	{attribute 'TcIecLibraryType'}
	{attribute 'external_name' := 'F_VN_PadImageBorderExp_GUID_A5E5D530_2DE0_2D11_697F_7D2919245E82'}
	(* Add padding around the original image borders. (expert function) *)
	FUNCTION F_VN_PadImageBorderExp : HRESULT
	VAR_INPUT
		ipSrcImage	:	ITcVnImage;	(* Source image *)
		ipPaddedImage	:	REFERENCE TO ITcVnImage;	(* Padded destination image (Same type as ipSrcImage, an appropriate destination image will be created if required.) *)
		nTopBorder	:	UDINT;	(* Padding height in pixels above top border *)
		nBottomBorder	:	UDINT;	(* Padding height in pixels below bottom border *)
		nLeftBorder	:	UDINT;	(* Padding width in pixels before left border *)
		nRightBorder	:	UDINT;	(* Padding width in pixels after right border *)
		ePaddingType	:	ETcVnBorderInterpolationMethod;	(* Specifies how the pixel values of the padding area are determined *)
	END_VAR
	VAR_IN_OUT
		aPaddingValue	:	TcVnVector4_LREAL;	(* Specifies the padding value if CONSTANT is used *)
	END_VAR
	VAR_INPUT
		hrPrev	:	HRESULT;	(* HRESULT indicating the result of previous operations (If SUCCEEDED(hrPrev) equals false, no operation is executed.) *)
	END_VAR

END_FUNCTION

// Functions/Basic Image Operations/F_VN_ReinterpretUnsupportedImage

	{attribute 'TcIecLibraryType'}
	{attribute 'external_name' := 'F_VN_ReinterpretUnsupportedImage_GUID_9CD6B2BD_CBC3_29A4_6E5B_0352FEEB17E8'}
	(* Reinterpret an unsupported image using additional information. If successful, the image will be of a supported type. *)
	FUNCTION F_VN_ReinterpretUnsupportedImage : HRESULT
	VAR_INPUT
		ipImage	:	ITcVnImage;	(* Image to be reinterpreted *)
		ePixelType	:	ETcVnElementType;	(* Pixel element type to be used for reinterpreting the image data *)
		hrPrev	:	HRESULT;	(* HRESULT indicating the result of previous operations (If SUCCEEDED(hrPrev) equals false, no operation is executed.) *)
	END_VAR

END_FUNCTION

// Functions/Basic Image Operations/F_VN_ResetRoi

	{attribute 'TcIecLibraryType'}
	{attribute 'external_name' := 'F_VN_ResetRoi_GUID_2C50FDC2_0370_20BD_7F54_98DAB1E9EC31'}
	(* Reset the region of interest (ROI) of an image. (After this operation, the ROI is set to the entire image.) *)
	FUNCTION F_VN_ResetRoi : HRESULT
	VAR_INPUT
		ipImage	:	ITcVnImage;	(* Image *)
		hrPrev	:	HRESULT;	(* HRESULT indicating the result of previous operations (If SUCCEEDED(hrPrev) equals false, no operation is executed.) *)
	END_VAR

END_FUNCTION

// Functions/Basic Image Operations/F_VN_SetImageChannel

	{attribute 'TcIecLibraryType'}
	{attribute 'external_name' := 'F_VN_SetImageChannel_GUID_0A11D43B_5EFB_299D_5725_A1931D902C34'}
	(* Sets the specified destination image channel to the values of the specified source image channel. *)
	FUNCTION F_VN_SetImageChannel : HRESULT
	VAR_INPUT
		ipSrcImage	:	ITcVnImage;	(* Source image *)
		ipDestImage	:	REFERENCE TO ITcVnImage;	(* Destination image (An appropriate image will be created if required.) *)
		nSrcChannelIndex	:	UINT;	(* Index of the source image channel *)
		nDestChannelIndex	:	UINT;	(* Index of the destination image channel, which will be replaced by the specified source image channel *)
		hrPrev	:	HRESULT;	(* HRESULT indicating the result of previous operations (If SUCCEEDED(hrPrev) equals false, no operation is executed.) *)
	END_VAR

END_FUNCTION

// Functions/Basic Image Operations/F_VN_SetPixel

	{attribute 'TcIecLibraryType'}
	{attribute 'external_name' := 'F_VN_SetPixel_GUID_8B44FC22_04B7_2DC7_7023_0AD245DB3507'}
	(* Sets a specific pixel. *)
	FUNCTION F_VN_SetPixel : HRESULT
	VAR_INPUT
		ipSrcImage	:	ITcVnImage;	(* Source image *)
	END_VAR
	VAR_IN_OUT
		aValue	:	TcVnVector4_LREAL;	(* The pixel value to set (additional channels are ignored.) *)
	END_VAR
	VAR_INPUT
		nX	:	UDINT;	(* x coordinate of the pixel *)
		nY	:	UDINT;	(* y coordinate of the pixel *)
		hrPrev	:	HRESULT;	(* HRESULT indicating the result of previous operations (If SUCCEEDED(hrPrev) equals false, no operation is executed.) *)
	END_VAR

END_FUNCTION

// Functions/Basic Image Operations/F_VN_SetPixels

	{attribute 'TcIecLibraryType'}
	{attribute 'external_name' := 'F_VN_SetPixels_GUID_FAE3DEC6_6066_2303_76C8_108C64D81E38'}
	(* Sets all pixels of an image to a given value. *)
	FUNCTION F_VN_SetPixels : HRESULT
	VAR_INPUT
		ipDestImage	:	ITcVnImage;	(* Destination image *)
	END_VAR
	VAR_IN_OUT
		aValue	:	TcVnVector4_LREAL;	(* Pixel value *)
	END_VAR
	VAR_INPUT
		hrPrev	:	HRESULT;	(* HRESULT indicating the result of previous operations (If SUCCEEDED(hrPrev) equals false, no operation is executed.) *)
	END_VAR

END_FUNCTION

// Functions/Basic Image Operations/F_VN_SetPixelsExp

	{attribute 'TcIecLibraryType'}
	{attribute 'external_name' := 'F_VN_SetPixelsExp_GUID_45CBC089_464B_2FAF_6251_E594A25ABBA2'}
	(* Sets all pixels of an image to a given value. (expert function) *)
	FUNCTION F_VN_SetPixelsExp : HRESULT
	VAR_INPUT
		ipDestImage	:	ITcVnImage;	(* Destination image *)
	END_VAR
	VAR_IN_OUT
		aValue	:	TcVnVector4_LREAL;	(* Pixel value *)
	END_VAR
	VAR_INPUT
		ipMask	:	ITcVnImage;	(* Mask image *)
		hrPrev	:	HRESULT;	(* HRESULT indicating the result of previous operations (If SUCCEEDED(hrPrev) equals false, no operation is executed.) *)
	END_VAR

END_FUNCTION

// Functions/Basic Image Operations/F_VN_SetRoi

	{attribute 'TcIecLibraryType'}
	{attribute 'external_name' := 'F_VN_SetRoi_GUID_6B5F6ACC_D699_29DC_6ACC_234995C24602'}
	(* Sets a region of interest (ROI) within an image. *)
	FUNCTION F_VN_SetRoi : HRESULT
	VAR_INPUT
		nX	:	UDINT;	(* Left boundary (inclusive 0-based index) *)
		nY	:	UDINT;	(* Upper boundary (inclusive 0-based index) *)
		nWidth	:	UDINT;	(* ROI width *)
		nHeight	:	UDINT;	(* ROI height *)
		ipDestImage	:	ITcVnImage;	(* Destination image *)
		hrPrev	:	HRESULT;	(* HRESULT indicating the result of previous operations (If SUCCEEDED(hrPrev) equals false, no operation is executed.) *)
	END_VAR

END_FUNCTION

// Functions/Basic Image Operations/F_VN_SetRoi_TcVnRectangle_DINT

	{attribute 'TcIecLibraryType'}
	{attribute 'external_name' := 'F_VN_SetRoi_TcVnRectangle_DINT_GUID_351427E6_8825_2F16_7392_DBA0A93C3EA1'}
	(* Sets a region of interest (ROI) within an image. *)
	FUNCTION F_VN_SetRoi_TcVnRectangle_DINT : HRESULT
	VAR_IN_OUT
		stRoi	:	TcVnRectangle_DINT;	(* Region of interest *)
	END_VAR
	VAR_INPUT
		ipDestImage	:	ITcVnImage;	(* Destination image *)
		hrPrev	:	HRESULT;	(* HRESULT indicating the result of previous operations (If SUCCEEDED(hrPrev) equals false, no operation is executed.) *)
	END_VAR

END_FUNCTION

// Functions/Basic Image Operations/F_VN_SetRoi_TcVnRectangle_UDINT

	{attribute 'TcIecLibraryType'}
	{attribute 'external_name' := 'F_VN_SetRoi_TcVnRectangle_UDINT_GUID_602E64BE_2371_25A7_7431_0AE2E6733D33'}
	(* Sets a region of interest (ROI) within an image. *)
	FUNCTION F_VN_SetRoi_TcVnRectangle_UDINT : HRESULT
	VAR_IN_OUT
		stRoi	:	TcVnRectangle_UDINT;	(* Region of interest *)
	END_VAR
	VAR_INPUT
		ipDestImage	:	ITcVnImage;	(* Destination image *)
		hrPrev	:	HRESULT;	(* HRESULT indicating the result of previous operations (If SUCCEEDED(hrPrev) equals false, no operation is executed.) *)
	END_VAR

END_FUNCTION

// Functions/Basic Image Operations/F_VN_SplitImageChannels

	{attribute 'TcIecLibraryType'}
	{attribute 'external_name' := 'F_VN_SplitImageChannels_GUID_A95E5FB7_F301_2632_66A4_8427D601C7CB'}
	(* Split a multi-channel image into multiple single channel images (1 for each source image channel). *)
	FUNCTION F_VN_SplitImageChannels : HRESULT
	VAR_INPUT
		ipSrcImage	:	ITcVnImage;	(* Source image with multiple channels *)
		pDestImages	:	PVOID;	(* Pointer to an array of ITcVnImage (appropriate destination images will be created if required) *)
		nArraySize	:	UINT;	(* Number of pDestImages array elements (array must be >= ipSourceImage channels) *)
		hrPrev	:	HRESULT;	(* HRESULT indicating the result of previous operations (If SUCCEEDED(hrPrev) equals false, no operation is executed.) *)
	END_VAR
	VAR_OUTPUT
		nImageChannels	:	UINT;	(* Actual source image channels *)
	END_VAR

END_FUNCTION

// Functions/Basic Image Operations/F_VN_TransformIntoDisplayableImageExp

	{attribute 'TcIecLibraryType'}
	{attribute 'external_name' := 'F_VN_TransformIntoDisplayableImageExp_GUID_167A9D9F_1F20_2D5B_6C90_35CDA27FBBBC'}
	(* Transform an image into a displayable image. The source image will be released and zeroed while existing destination images will be released and overwritten with the function result. If bAllowDeepCopy equals false, the source image must not be used anywhere else and the transformation is always very fast. Otherwise, if bAllowDeepCopy equals true, a deep copy of the source image might be created if required, which will result in a longer execution time. If you want to use ipSrcImage after this function call, use F_VN_CopyIntoDisplayableImage instead. (expert function) *)
	FUNCTION F_VN_TransformIntoDisplayableImageExp : HRESULT
	VAR_INPUT
		ipSrcImage	:	REFERENCE TO ITcVnImage;	(* Source image *)
		ipDestImage	:	REFERENCE TO ITcVnDisplayableImage;	(* Returns the displayable image *)
		bAllowDeepCopy	:	BOOL;	(* Allow deep image copies, if required *)
		hrPrev	:	HRESULT;	(* HRESULT indicating the result of previous operations (If SUCCEEDED(hrPrev) equals false, no operation is executed.) *)
	END_VAR

END_FUNCTION

// Functions/Container Statistics/F_VN_ContainerAverage

	{attribute 'TcIecLibraryType'}
	{attribute 'external_name' := 'F_VN_ContainerAverage_GUID_AA883F39_9BF3_2D50_47D7_60462300CF21'}
	(* Calculate the average of elements in a container. *)
	FUNCTION F_VN_ContainerAverage : HRESULT
	VAR_INPUT
		ipSrcContainer	:	ITcVnContainer;	(* Source container (Arithmetic, point and vector element types are supported. For points and vectors, the euclidean norm is used.) *)
	END_VAR
	VAR_IN_OUT
		fAverage	:	LREAL;	(* Returns the calculated average value *)
	END_VAR
	VAR_INPUT
		hrPrev	:	HRESULT;	(* HRESULT indicating the result of previous operations (If SUCCEEDED(hrPrev) equals false, no operation is executed.) *)
	END_VAR

END_FUNCTION

// Functions/Container Statistics/F_VN_ContainerAverageElementwise2

	{attribute 'TcIecLibraryType'}
	{attribute 'external_name' := 'F_VN_ContainerAverageElementwise2_GUID_A5968F66_4B6A_2FA7_4E6D_E4702B7B6763'}
	(* Calculate the elementwise average of 2D elements in a container. *)
	FUNCTION F_VN_ContainerAverageElementwise2 : HRESULT
	VAR_INPUT
		ipSrcContainer	:	ITcVnContainer;	(* Source container with 2D points or vectors *)
	END_VAR
	VAR_IN_OUT
		aAverage	:	TcVnVector2_LREAL;	(* Returns the calculated average values *)
	END_VAR
	VAR_INPUT
		hrPrev	:	HRESULT;	(* HRESULT indicating the result of previous operations (If SUCCEEDED(hrPrev) equals false, no operation is executed.) *)
	END_VAR

END_FUNCTION

// Functions/Container Statistics/F_VN_ContainerAverageElementwise3

	{attribute 'TcIecLibraryType'}
	{attribute 'external_name' := 'F_VN_ContainerAverageElementwise3_GUID_40FE5448_4613_25F6_6B44_B58BBFE3E301'}
	(* Calculate the elementwise average of 3D elements in a container. *)
	FUNCTION F_VN_ContainerAverageElementwise3 : HRESULT
	VAR_INPUT
		ipSrcContainer	:	ITcVnContainer;	(* Source container with 3D points or vectors *)
	END_VAR
	VAR_IN_OUT
		aAverage	:	TcVnVector3_LREAL;	(* Returns the calculated average values *)
	END_VAR
	VAR_INPUT
		hrPrev	:	HRESULT;	(* HRESULT indicating the result of previous operations (If SUCCEEDED(hrPrev) equals false, no operation is executed.) *)
	END_VAR

END_FUNCTION

// Functions/Container Statistics/F_VN_ContainerAverageElementwise4

	{attribute 'TcIecLibraryType'}
	{attribute 'external_name' := 'F_VN_ContainerAverageElementwise4_GUID_DEACFB72_F4A2_2C02_42D9_1C2A0DD59263'}
	(* Calculate the elementwise average of 4D elements in a container. *)
	FUNCTION F_VN_ContainerAverageElementwise4 : HRESULT
	VAR_INPUT
		ipSrcContainer	:	ITcVnContainer;	(* Source container with 4D vectors *)
	END_VAR
	VAR_IN_OUT
		aAverage	:	TcVnVector4_LREAL;	(* Returns the calculated average values *)
	END_VAR
	VAR_INPUT
		hrPrev	:	HRESULT;	(* HRESULT indicating the result of previous operations (If SUCCEEDED(hrPrev) equals false, no operation is executed.) *)
	END_VAR

END_FUNCTION

// Functions/Container Statistics/F_VN_ContainerAverageVariance

	{attribute 'TcIecLibraryType'}
	{attribute 'external_name' := 'F_VN_ContainerAverageVariance_GUID_F86D5373_0B69_212E_4923_C1F41E37B181'}
	(* Calculate the average and variance of elements in a container. *)
	FUNCTION F_VN_ContainerAverageVariance : HRESULT
	VAR_INPUT
		ipSrcContainer	:	ITcVnContainer;	(* Source container (Arithmetic, point and vector element types are supported. For points and vectors, the euclidean norm is used.) *)
	END_VAR
	VAR_IN_OUT
		fAverage	:	LREAL;	(* Returns the calculated average value *)
		fVariance	:	LREAL;	(* Returns the calculated variance value *)
	END_VAR
	VAR_INPUT
		hrPrev	:	HRESULT;	(* HRESULT indicating the result of previous operations (If SUCCEEDED(hrPrev) equals false, no operation is executed.) *)
	END_VAR

END_FUNCTION

// Functions/Container Statistics/F_VN_ContainerAverageVarianceElementwise2

	{attribute 'TcIecLibraryType'}
	{attribute 'external_name' := 'F_VN_ContainerAverageVarianceElementwise2_GUID_9DD8D138_D087_2ADB_447F_BCA5C1C4B858'}
	(* Calculate the elementwise average and variance of 2D elements in a container. *)
	FUNCTION F_VN_ContainerAverageVarianceElementwise2 : HRESULT
	VAR_INPUT
		ipSrcContainer	:	ITcVnContainer;	(* Source container with 2D points or vectors *)
	END_VAR
	VAR_IN_OUT
		aAverage	:	TcVnVector2_LREAL;	(* Returns the calculated average values *)
		aVariance	:	TcVnVector2_LREAL;	(* Returns the calculated variance values *)
	END_VAR
	VAR_INPUT
		hrPrev	:	HRESULT;	(* HRESULT indicating the result of previous operations (If SUCCEEDED(hrPrev) equals false, no operation is executed.) *)
	END_VAR

END_FUNCTION

// Functions/Container Statistics/F_VN_ContainerAverageVarianceElementwise3

	{attribute 'TcIecLibraryType'}
	{attribute 'external_name' := 'F_VN_ContainerAverageVarianceElementwise3_GUID_FA835F97_60F3_2236_51E3_712391145764'}
	(* Calculate the elementwise average and variance of 3D elements in a container. *)
	FUNCTION F_VN_ContainerAverageVarianceElementwise3 : HRESULT
	VAR_INPUT
		ipSrcContainer	:	ITcVnContainer;	(* Source container with 3D points or vectors *)
	END_VAR
	VAR_IN_OUT
		aAverage	:	TcVnVector3_LREAL;	(* Returns the calculated average values *)
		aVariance	:	TcVnVector3_LREAL;	(* Returns the calculated variance values *)
	END_VAR
	VAR_INPUT
		hrPrev	:	HRESULT;	(* HRESULT indicating the result of previous operations (If SUCCEEDED(hrPrev) equals false, no operation is executed.) *)
	END_VAR

END_FUNCTION

// Functions/Container Statistics/F_VN_ContainerAverageVarianceElementwise4

	{attribute 'TcIecLibraryType'}
	{attribute 'external_name' := 'F_VN_ContainerAverageVarianceElementwise4_GUID_031E1C0B_D296_2CEF_785B_2052A4B44928'}
	(* Calculate the elementwise average and variance of 4D elements in a container. *)
	FUNCTION F_VN_ContainerAverageVarianceElementwise4 : HRESULT
	VAR_INPUT
		ipSrcContainer	:	ITcVnContainer;	(* Source container with 4D vectors *)
	END_VAR
	VAR_IN_OUT
		aAverage	:	TcVnVector4_LREAL;	(* Returns the calculated average values *)
		aVariance	:	TcVnVector4_LREAL;	(* Returns the calculated variance values *)
	END_VAR
	VAR_INPUT
		hrPrev	:	HRESULT;	(* HRESULT indicating the result of previous operations (If SUCCEEDED(hrPrev) equals false, no operation is executed.) *)
	END_VAR

END_FUNCTION

// Functions/Container Statistics/F_VN_MaxElement

	{attribute 'TcIecLibraryType'}
	{attribute 'external_name' := 'F_VN_MaxElement_GUID_9353BD58_8969_23CD_6837_1D5672DD3636'}
	(* Gets the maximum element of a container. *)
	FUNCTION F_VN_MaxElement : HRESULT
	VAR_INPUT
		ipSrcContainer	:	ITcVnContainer;	(* Source container (Arithmetic, point and vector element types are supported. For points and vectors, the euclidean norm is used.) *)
		ipDestIterator	:	REFERENCE TO ITcVnBidirectionalIterator;	(* Returns an iterator to the requested element *)
	END_VAR
	VAR_IN_OUT
		nIndex	:	ULINT;	(* Returns the position of the requested element within the container *)
	END_VAR
	VAR_INPUT
		hrPrev	:	HRESULT;	(* HRESULT indicating the result of previous operations (If SUCCEEDED(hrPrev) equals false, no operation is executed.) *)
	END_VAR

END_FUNCTION

// Functions/Container Statistics/F_VN_MedianElement

	{attribute 'TcIecLibraryType'}
	{attribute 'external_name' := 'F_VN_MedianElement_GUID_734602DB_9D28_2D88_734A_BDC3C8FE153F'}
	(* Gets the median element of a container. *)
	FUNCTION F_VN_MedianElement : HRESULT
	VAR_INPUT
		ipSrcContainer	:	ITcVnContainer;	(* Source container (Arithmetic, point and vector element types are supported. For points and vectors, the euclidean norm is used.) *)
		ipDestIterator	:	REFERENCE TO ITcVnBidirectionalIterator;	(* Returns an iterator to the requested element *)
	END_VAR
	VAR_IN_OUT
		nIndex	:	ULINT;	(* Returns the position of the requested element within the container *)
	END_VAR
	VAR_INPUT
		hrPrev	:	HRESULT;	(* HRESULT indicating the result of previous operations (If SUCCEEDED(hrPrev) equals false, no operation is executed.) *)
	END_VAR

END_FUNCTION

// Functions/Container Statistics/F_VN_MinElement

	{attribute 'TcIecLibraryType'}
	{attribute 'external_name' := 'F_VN_MinElement_GUID_9563E038_8D44_21FD_4C05_B15238CF2018'}
	(* Gets the minimum element of a container. *)
	FUNCTION F_VN_MinElement : HRESULT
	VAR_INPUT
		ipSrcContainer	:	ITcVnContainer;	(* Source container (Arithmetic, point and vector element types are supported. For points and vectors, the euclidean norm is used.) *)
		ipDestIterator	:	REFERENCE TO ITcVnBidirectionalIterator;	(* Returns an iterator to the requested element *)
	END_VAR
	VAR_IN_OUT
		nIndex	:	ULINT;	(* Returns the position of the requested element within the container *)
	END_VAR
	VAR_INPUT
		hrPrev	:	HRESULT;	(* HRESULT indicating the result of previous operations (If SUCCEEDED(hrPrev) equals false, no operation is executed.) *)
	END_VAR

END_FUNCTION

// Functions/Fourier Analysis/F_VN_CreateBandpassButterworthFilter

	{attribute 'TcIecLibraryType'}
	{attribute 'external_name' := 'F_VN_CreateBandpassButterworthFilter_GUID_A4719FC8_3078_205C_4E26_9139901FC7B0'}
	(* Creates a bandpass Butterworth filter, which can be applied to a frequency domain image by element-wise multiplication. *)
	FUNCTION F_VN_CreateBandpassButterworthFilter : HRESULT
	VAR_INPUT
		ipFilter	:	REFERENCE TO ITcVnImage;	(* Returns the created filter (1 channel of type REAL or LREAL, depending on bDoublePrecision. Non-zero interface pointers are reused.). *)
		nWidth	:	UDINT;	(* Filter width (even, >= 2, must match the width of the image it is applied to) *)
		nHeight	:	UDINT;	(* Filter height (even, >= 2, must match the height of the image it is applied to) *)
		bDoublePrecision	:	BOOL;	(* If true, the filter is generated with double precision (LREAL) instead of single precision (REAL). *)
		bOriginAtCenter	:	BOOL;	(* If true, the filter origin is shifted to the image center. *)
		fCutoffDistance	:	LREAL;	(* The cutoff distance of the Butterworth filter (> 0). *)
		fBandWidth	:	LREAL;	(* The band width of the Butterworth filter (> 0). *)
		nOrder	:	UDINT;	(* The order of the Butterworth filter (> 0). *)
		fScale	:	LREAL;	(* The scale factor of the Butterworth filter denominator term (> 0, e.g. 0.414 or 1.0). *)
		hrPrev	:	HRESULT;	(* HRESULT indicating the result of previous operations (If SUCCEEDED(hrPrev) equals false, no operation is executed.) *)
	END_VAR

END_FUNCTION

// Functions/Fourier Analysis/F_VN_CreateBandpassGaussianFilter

	{attribute 'TcIecLibraryType'}
	{attribute 'external_name' := 'F_VN_CreateBandpassGaussianFilter_GUID_AB3E0B05_028B_2322_7CF4_87504E4D004F'}
	(* Creates a bandpass Gaussian filter, which can be applied to a frequency domain image by element-wise multiplication. *)
	FUNCTION F_VN_CreateBandpassGaussianFilter : HRESULT
	VAR_INPUT
		ipFilter	:	REFERENCE TO ITcVnImage;	(* Returns the created filter (1 channel of type REAL or LREAL, depending on bDoublePrecision. Non-zero interface pointers are reused.). *)
		nWidth	:	UDINT;	(* Filter width (even, >= 2, must match the width of the image it is applied to) *)
		nHeight	:	UDINT;	(* Filter height (even, >= 2, must match the height of the image it is applied to) *)
		bDoublePrecision	:	BOOL;	(* If true, the filter is generated with double precision (LREAL) instead of single precision (REAL). *)
		bOriginAtCenter	:	BOOL;	(* If true, the filter origin is shifted to the image center. *)
		fCutoffDistance	:	LREAL;	(* The cutoff distance of the Gaussian filter (> 0). *)
		fBandWidth	:	LREAL;	(* The band width of the Gaussian filter (> 0). *)
		hrPrev	:	HRESULT;	(* HRESULT indicating the result of previous operations (If SUCCEEDED(hrPrev) equals false, no operation is executed.) *)
	END_VAR

END_FUNCTION

// Functions/Fourier Analysis/F_VN_CreateBandrejectButterworthFilter

	{attribute 'TcIecLibraryType'}
	{attribute 'external_name' := 'F_VN_CreateBandrejectButterworthFilter_GUID_43FD0880_9A03_21BB_62EE_0C372A51F6F1'}
	(* Creates a bandreject Butterworth filter, which can be applied to a frequency domain image by element-wise multiplication. *)
	FUNCTION F_VN_CreateBandrejectButterworthFilter : HRESULT
	VAR_INPUT
		ipFilter	:	REFERENCE TO ITcVnImage;	(* Returns the created filter (1 channel of type REAL or LREAL, depending on bDoublePrecision. Non-zero interface pointers are reused.). *)
		nWidth	:	UDINT;	(* Filter width (even, >= 2, must match the width of the image it is applied to) *)
		nHeight	:	UDINT;	(* Filter height (even, >= 2, must match the height of the image it is applied to) *)
		bDoublePrecision	:	BOOL;	(* If true, the filter is generated with double precision (LREAL) instead of single precision (REAL). *)
		bOriginAtCenter	:	BOOL;	(* If true, the filter origin is shifted to the image center. *)
		fCutoffDistance	:	LREAL;	(* The cutoff distance of the Butterworth filter (> 0). *)
		fBandWidth	:	LREAL;	(* The band width of the Butterworth filter (> 0). *)
		nOrder	:	UDINT;	(* The order of the Butterworth filter (> 0). *)
		fScale	:	LREAL;	(* The scale factor of the Butterworth filter denominator term (> 0, e.g. 0.414 or 1.0). *)
		hrPrev	:	HRESULT;	(* HRESULT indicating the result of previous operations (If SUCCEEDED(hrPrev) equals false, no operation is executed.) *)
	END_VAR

END_FUNCTION

// Functions/Fourier Analysis/F_VN_CreateBandrejectGaussianFilter

	{attribute 'TcIecLibraryType'}
	{attribute 'external_name' := 'F_VN_CreateBandrejectGaussianFilter_GUID_2D030AC7_64BE_238B_728C_49B2827F9032'}
	(* Creates a bandreject Gaussian filter, which can be applied to a frequency domain image by element-wise multiplication. *)
	FUNCTION F_VN_CreateBandrejectGaussianFilter : HRESULT
	VAR_INPUT
		ipFilter	:	REFERENCE TO ITcVnImage;	(* Returns the created filter (1 channel of type REAL or LREAL, depending on bDoublePrecision. Non-zero interface pointers are reused.). *)
		nWidth	:	UDINT;	(* Filter width (even, >= 2, must match the width of the image it is applied to) *)
		nHeight	:	UDINT;	(* Filter height (even, >= 2, must match the height of the image it is applied to) *)
		bDoublePrecision	:	BOOL;	(* If true, the filter is generated with double precision (LREAL) instead of single precision (REAL). *)
		bOriginAtCenter	:	BOOL;	(* If true, the filter origin is shifted to the image center. *)
		fCutoffDistance	:	LREAL;	(* The cutoff distance of the Gaussian filter (> 0). *)
		fBandWidth	:	LREAL;	(* The band width of the Gaussian filter (> 0). *)
		hrPrev	:	HRESULT;	(* HRESULT indicating the result of previous operations (If SUCCEEDED(hrPrev) equals false, no operation is executed.) *)
	END_VAR

END_FUNCTION

// Functions/Fourier Analysis/F_VN_CreateHighpassButterworthFilter

	{attribute 'TcIecLibraryType'}
	{attribute 'external_name' := 'F_VN_CreateHighpassButterworthFilter_GUID_26315EFD_6407_2DDF_6510_E1ECDEDCA359'}
	(* Creates a highpass Butterworth filter, which can be applied to a frequency domain image by element-wise multiplication. *)
	FUNCTION F_VN_CreateHighpassButterworthFilter : HRESULT
	VAR_INPUT
		ipFilter	:	REFERENCE TO ITcVnImage;	(* Returns the created filter (1 channel of type REAL or LREAL, depending on bDoublePrecision. Non-zero interface pointers are reused.). *)
		nWidth	:	UDINT;	(* Filter width (even, >= 2, must match the width of the image it is applied to) *)
		nHeight	:	UDINT;	(* Filter height (even, >= 2, must match the height of the image it is applied to) *)
		bDoublePrecision	:	BOOL;	(* If true, the filter is generated with double precision (LREAL) instead of single precision (REAL). *)
		bOriginAtCenter	:	BOOL;	(* If true, the filter origin is shifted to the image center. *)
		fCutoffDistance	:	LREAL;	(* The cutoff distance of the Butterworth filter (> 0). *)
		nOrder	:	UDINT;	(* The order of the Butterworth filter (> 0). *)
		fScale	:	LREAL;	(* The scale factor of the Butterworth filter denominator term (> 0, e.g. 0.414 or 1.0). *)
		hrPrev	:	HRESULT;	(* HRESULT indicating the result of previous operations (If SUCCEEDED(hrPrev) equals false, no operation is executed.) *)
	END_VAR

END_FUNCTION

// Functions/Fourier Analysis/F_VN_CreateHighpassGaussianFilter

	{attribute 'TcIecLibraryType'}
	{attribute 'external_name' := 'F_VN_CreateHighpassGaussianFilter_GUID_91B5C0DC_EE24_21D2_4440_C5D5A4FE32A8'}
	(* Creates a highpass Gaussian filter, which can be applied to a frequency domain image by element-wise multiplication. *)
	FUNCTION F_VN_CreateHighpassGaussianFilter : HRESULT
	VAR_INPUT
		ipFilter	:	REFERENCE TO ITcVnImage;	(* Returns the created filter (1 channel of type REAL or LREAL, depending on bDoublePrecision. Non-zero interface pointers are reused.). *)
		nWidth	:	UDINT;	(* Filter width (even, >= 2, must match the width of the image it is applied to) *)
		nHeight	:	UDINT;	(* Filter height (even, >= 2, must match the height of the image it is applied to) *)
		bDoublePrecision	:	BOOL;	(* If true, the filter is generated with double precision (LREAL) instead of single precision (REAL). *)
		bOriginAtCenter	:	BOOL;	(* If true, the filter origin is shifted to the image center. *)
		fCutoffDistance	:	LREAL;	(* The cutoff distance of the Gaussian filter (> 0). *)
		hrPrev	:	HRESULT;	(* HRESULT indicating the result of previous operations (If SUCCEEDED(hrPrev) equals false, no operation is executed.) *)
	END_VAR

END_FUNCTION

// Functions/Fourier Analysis/F_VN_CreateLowpassButterworthFilter

	{attribute 'TcIecLibraryType'}
	{attribute 'external_name' := 'F_VN_CreateLowpassButterworthFilter_GUID_373093B4_3E27_26A4_696A_3EE89B988877'}
	(* Creates a lowpass Butterworth filter, which can be applied to a frequency domain image by element-wise multiplication. *)
	FUNCTION F_VN_CreateLowpassButterworthFilter : HRESULT
	VAR_INPUT
		ipFilter	:	REFERENCE TO ITcVnImage;	(* Returns the created filter (1 channel of type REAL or LREAL, depending on bDoublePrecision. Non-zero interface pointers are reused.). *)
		nWidth	:	UDINT;	(* Filter width (even, >= 2, must match the width of the image it is applied to) *)
		nHeight	:	UDINT;	(* Filter height (even, >= 2, must match the height of the image it is applied to) *)
		bDoublePrecision	:	BOOL;	(* If true, the filter is generated with double precision (LREAL) instead of single precision (REAL). *)
		bOriginAtCenter	:	BOOL;	(* If true, the filter origin is shifted to the image center. *)
		fCutoffDistance	:	LREAL;	(* The cutoff distance of the Butterworth filter (> 0). *)
		nOrder	:	UDINT;	(* The order of the Butterworth filter (> 0). *)
		fScale	:	LREAL;	(* The scale factor of the Butterworth filter denominator term (> 0, e.g. 0.414 or 1.0). *)
		hrPrev	:	HRESULT;	(* HRESULT indicating the result of previous operations (If SUCCEEDED(hrPrev) equals false, no operation is executed.) *)
	END_VAR

END_FUNCTION

// Functions/Fourier Analysis/F_VN_CreateLowpassGaussianFilter

	{attribute 'TcIecLibraryType'}
	{attribute 'external_name' := 'F_VN_CreateLowpassGaussianFilter_GUID_FC365988_00B2_289F_4A02_DA34E2899A69'}
	(* Creates a lowpass Gaussian filter, which can be applied to a frequency domain image by element-wise multiplication. *)
	FUNCTION F_VN_CreateLowpassGaussianFilter : HRESULT
	VAR_INPUT
		ipFilter	:	REFERENCE TO ITcVnImage;	(* Returns the created filter (1 channel of type REAL or LREAL, depending on bDoublePrecision. Non-zero interface pointers are reused.). *)
		nWidth	:	UDINT;	(* Filter width (even, >= 2, must match the width of the image it is applied to) *)
		nHeight	:	UDINT;	(* Filter height (even, >= 2, must match the height of the image it is applied to) *)
		bDoublePrecision	:	BOOL;	(* If true, the filter is generated with double precision (LREAL) instead of single precision (REAL). *)
		bOriginAtCenter	:	BOOL;	(* If true, the filter origin is shifted to the image center. *)
		fCutoffDistance	:	LREAL;	(* The cutoff distance of the Gaussian filter (> 0). *)
		hrPrev	:	HRESULT;	(* HRESULT indicating the result of previous operations (If SUCCEEDED(hrPrev) equals false, no operation is executed.) *)
	END_VAR

END_FUNCTION

// Functions/Fourier Analysis/F_VN_Dft

	{attribute 'TcIecLibraryType'}
	{attribute 'external_name' := 'F_VN_Dft_GUID_9CD2E68A_8224_2AA6_4C68_735CDE258796'}
	(* Computes the DFT for a given image. *)
	FUNCTION F_VN_Dft : HRESULT
	VAR_INPUT
		ipSpatialImage	:	ITcVnImage;	(* Source image (elements of type REAL or LREAL, 1 (Re) or 2 (Re + Im) channels) *)
		ipFrequencyImage	:	REFERENCE TO ITcVnImage;	(* Destination image (same type as ipSpatialImage, but number of channels and size can vary depending on bPackedCCS and bAutoPadding. *)
		bPackedCCS	:	BOOL;	(* If true and ipSpatialImage has only 1 channel, the result image will have 1 channel with packed complex-conjugate-symmetrical format results. Otherwise, the result image will have 2 separate channels (Re + Im), containing the full spectrum. *)
		bAutoPadding	:	BOOL;	(* If true, the input image is automatically padded (with 0s) to optimal size if required, to speed up dft (Creates a temporary copy so that ipSpatialImage content stays unchanged, which also requires some additional computation power. Therefore, it is recommended to compare execution times with and without padding.) *)
		hrPrev	:	HRESULT;	(* HRESULT indicating the result of previous operations (If SUCCEEDED(hrPrev) equals false, no operation is executed.) *)
	END_VAR

END_FUNCTION

// Functions/Fourier Analysis/F_VN_InverseDft

	{attribute 'TcIecLibraryType'}
	{attribute 'external_name' := 'F_VN_InverseDft_GUID_5190C4B2_3FA3_2B1D_6D96_EBC870B13024'}
	(* Compute the inverse DFT for a given frequency image. *)
	FUNCTION F_VN_InverseDft : HRESULT
	VAR_INPUT
		ipFrequencyImage	:	ITcVnImage;	(* Source frequency image (elements of type REAL or LREAL, 1 (packed CCS) or 2 (Re + Im) channels) *)
		ipSpatialImage	:	REFERENCE TO ITcVnImage;	(* Destination image (Same type as ipFrequencyImage, but number of channels can vary depending on bRealOutput. An appropriate image will be created if required.) *)
		bRealOutput	:	BOOL;	(* Only relevant if ipFrequencyImage has 2 channels. If true, the result image will have only 1 channel. Otherwise, the result image will have 2 separate channels (Re + Im). If ipFrequencyImage has only 1 channel, packed CCS format is assumed and the result image will always have only 1 channel. *)
		hrPrev	:	HRESULT;	(* HRESULT indicating the result of previous operations (If SUCCEEDED(hrPrev) equals false, no operation is executed.) *)
	END_VAR

END_FUNCTION

// Functions/Fourier Analysis/F_VN_OptimalDftSize

	{attribute 'TcIecLibraryType'}
	{attribute 'external_name' := 'F_VN_OptimalDftSize_GUID_7F72AB5E_E31E_25EC_575C_20FDDD4E5230'}
	(* Computes the optimal image size for applying a dft (can lead to better performance). *)
	FUNCTION F_VN_OptimalDftSize : HRESULT
	VAR_INPUT
		ipImage	:	ITcVnImage;	(* Source image for which to compute the optimal width and height *)
	END_VAR
	VAR_IN_OUT
		nOptWidth	:	UDINT;	(* Returns the optimal width of the image *)
		nOptHeight	:	UDINT;	(* Returns the optimal height of the image *)
	END_VAR
	VAR_INPUT
		hrPrev	:	HRESULT;	(* HRESULT indicating the result of previous operations (If SUCCEEDED(hrPrev) equals false, no operation is executed.) *)
	END_VAR

END_FUNCTION

// Functions/Machine Learning/F_VN_CreateBoostClassifier

	{attribute 'TcIecLibraryType'}
	{attribute 'external_name' := 'F_VN_CreateBoostClassifier_GUID_DE956DB3_C6B5_20EF_6F40_CA0A52E7B053'}
	(* Create a Boost classifier using the default parameters. The initial reference count is set to one if a new model is created and kept, otherwise. The Boost classifier is only applicable to binary classification problems. It learns to distinguish between samples labelled with two user-defined class labels by incrementally adding weak classifiers to improve the classification results. Models of this type neither support on-line training (sample by sample) nor retraining. *)
	FUNCTION F_VN_CreateBoostClassifier : HRESULT
	VAR_INPUT
		ipMlModel	:	REFERENCE TO ITcVnMlModel;	(* Returns the created model (Non-zero interface pointers are reused.) *)
		hrPrev	:	HRESULT;	(* HRESULT indicating the result of previous operations (If SUCCEEDED(hrPrev) equals false, no operation is executed.) *)
	END_VAR

END_FUNCTION

// Functions/Machine Learning/F_VN_CreateBoostClassifierExp

	{attribute 'TcIecLibraryType'}
	{attribute 'external_name' := 'F_VN_CreateBoostClassifierExp_GUID_DBB0D30D_27D6_284A_7AD2_009715990AF3'}
	(* Create a Boost classifier. The initial reference count is set to one if a new model is created and kept, otherwise. The Boost classifier is only applicable to binary classification problems. It learns to distinguish between samples labelled with two user-defined class labels by incrementally adding weak classifiers to improve the classification results. Models of this type neither support on-line training (sample by sample) nor retraining. (expert function) *)
	FUNCTION F_VN_CreateBoostClassifierExp : HRESULT
	VAR_INPUT
		ipMlModel	:	REFERENCE TO ITcVnMlModel;	(* Returns the created model (Non-zero interface pointers are reused.) *)
		eType	:	ETcVnBoostClassifierType;	(* Learning algorithm type (default: TCVN_BCT_REAL) *)
		nMaxDepth	:	UDINT;	(* Maximum tree depth (default: 1) *)
		nMinSamples	:	UDINT;	(* Minimum number of samples within a node required for splitting (default: 10) *)
		nWeakClassifiers	:	UDINT;	(* Number of weak classifiers (default: 100) *)
		fWeightTrimRate	:	LREAL;	(* Weight threshold used during training (off: 0; default: 0.95). *)
		hrPrev	:	HRESULT;	(* HRESULT indicating the result of previous operations (If SUCCEEDED(hrPrev) equals false, no operation is executed.) *)
	END_VAR

END_FUNCTION

// Functions/Machine Learning/F_VN_CreateBoostClassifierExp2

	{attribute 'TcIecLibraryType'}
	{attribute 'external_name' := 'F_VN_CreateBoostClassifierExp2_GUID_6FAFAEAC_CC9F_2757_6896_43BC81C44B2C'}
	(* Create a Boost classifier. The initial reference count is set to one if a new model is created and kept, otherwise. The Boost classifier is only applicable to binary classification problems. It learns to distinguish between samples labelled with two user-defined class labels by incrementally adding weak classifiers to improve the classification results. Models of this type neither support on-line training (sample by sample) nor retraining. (expert function) *)
	FUNCTION F_VN_CreateBoostClassifierExp2 : HRESULT
	VAR_INPUT
		ipMlModel	:	REFERENCE TO ITcVnMlModel;	(* Returns the created model (Non-zero interface pointers are reused.) *)
		eType	:	ETcVnBoostClassifierType;	(* Learning algorithm type (default: TCVN_BCT_REAL) *)
		nMaxDepth	:	UDINT;	(* Maximum tree depth (default: 1) *)
		nMinSamples	:	UDINT;	(* Minimum number of samples within a node required for splitting (default: 10) *)
		nWeakClassifiers	:	UDINT;	(* Number of weak classifiers (default: 100) *)
		fWeightTrimRate	:	LREAL;	(* Weight threshold used during training (off: 0; default: 0.95). *)
		ipClassPriors	:	ITcVnContainer;	(* Class priors (ContainerType_Vector_REAL or ContainerType_Vector_LREAL; only for classifiers; optional, set to 0 if not required or not allowed; default: 0) *)
		hrPrev	:	HRESULT;	(* HRESULT indicating the result of previous operations (If SUCCEEDED(hrPrev) equals false, no operation is executed.) *)
	END_VAR

END_FUNCTION

// Functions/Machine Learning/F_VN_CreateKmppModel

	{attribute 'TcIecLibraryType'}
	{attribute 'external_name' := 'F_VN_CreateKmppModel_GUID_FC31DC4A_EF37_2F62_55C6_7F765B594AB6'}
	(* Create a k-means++ model of the specified type. The initial reference count is set to one if a new model is created and kept, otherwise. Models of this type neither support on-line training (sample by sample) nor retraining. *)
	FUNCTION F_VN_CreateKmppModel : HRESULT
	VAR_INPUT
		ipMlModel	:	REFERENCE TO ITcVnMlModel;	(* Returns the created model (Non-zero interface pointers are reused.) *)
		eKmppType	:	ETcVnPrototypeClusterer;	(* k-means++ model type *)
		nK	:	UDINT;	(* Parameter k (number of clusters) *)
		hrPrev	:	HRESULT;	(* HRESULT indicating the result of previous operations (If SUCCEEDED(hrPrev) equals false, no operation is executed.) *)
	END_VAR

END_FUNCTION

// Functions/Machine Learning/F_VN_CreateKmppModelExp

	{attribute 'TcIecLibraryType'}
	{attribute 'external_name' := 'F_VN_CreateKmppModelExp_GUID_91671E6C_0B95_2041_7EBD_EB43C5B888BE'}
	(* Create a k-means++ model of the specified type. The initial reference count is set to one if a new model is created and kept, otherwise. Models of this type neither support on-line training (sample by sample) nor retraining. (expert function) *)
	FUNCTION F_VN_CreateKmppModelExp : HRESULT
	VAR_INPUT
		ipMlModel	:	REFERENCE TO ITcVnMlModel;	(* Returns the created model (Non-zero interface pointers are reused.) *)
		eKmppType	:	ETcVnPrototypeClusterer;	(* k-means++ model type *)
		nK	:	UDINT;	(* Parameter k (number of clusters) *)
		bDoublePrecision	:	BOOL;	(* If true, the model is generated with double precision (LREAL) instead of single precision (REAL). (default: FALSE) *)
		nMaxIterations	:	UDINT;	(* Maximum number of iterations (triggers the usage of the default value of 10 if it equals 0) *)
		fEpsilon	:	LREAL;	(* Maximum allowed difference of the error between two successive iterations (triggers the usage of the default value of 0.001 if it equals 0) *)
		hrPrev	:	HRESULT;	(* HRESULT indicating the result of previous operations (If SUCCEEDED(hrPrev) equals false, no operation is executed.) *)
	END_VAR

END_FUNCTION

// Functions/Machine Learning/F_VN_CreateKnnModel

	{attribute 'TcIecLibraryType'}
	{attribute 'external_name' := 'F_VN_CreateKnnModel_GUID_3FC5A2A1_2868_235E_7F18_46CEDDCDBFFE'}
	(* Create a k-nearest neighbors model of the specified type. The initial reference count is set to one if a new model is created and kept, otherwise. Models of this type support on-line training (sample by sample) and retraining. Predictions can only be scalar. *)
	FUNCTION F_VN_CreateKnnModel : HRESULT
	VAR_INPUT
		ipMlModel	:	REFERENCE TO ITcVnMlModel;	(* Returns the created model (Non-zero interface pointers are reused.) *)
		eKnnType	:	ETcVnKnn;	(* k-nearest neighbors model type *)
		nK	:	UDINT;	(* Parameter k used for prediction (number of considered neighbors) *)
		hrPrev	:	HRESULT;	(* HRESULT indicating the result of previous operations (If SUCCEEDED(hrPrev) equals false, no operation is executed.) *)
	END_VAR

END_FUNCTION

// Functions/Machine Learning/F_VN_CreateLbgModel

	{attribute 'TcIecLibraryType'}
	{attribute 'external_name' := 'F_VN_CreateLbgModel_GUID_A89F132A_3261_218A_640A_D3FE962B6F46'}
	(* Create a LBG model of the specified type. The initial reference count is set to one if a new model is created and kept, otherwise. Models of this type neither support on-line training (sample by sample) nor retraining. *)
	FUNCTION F_VN_CreateLbgModel : HRESULT
	VAR_INPUT
		ipMlModel	:	REFERENCE TO ITcVnMlModel;	(* Returns the created model (Non-zero interface pointers are reused.) *)
		eLbgType	:	ETcVnPrototypeClusterer;	(* LBG model type *)
		nMaxClusters	:	UDINT;	(* Maximum number of clusters *)
		fMaxClusterRadius	:	LREAL;	(* Maximum allowed radius (L2 norm) of a single cluster, i.e. clusters with a higher radius will be split into smaller ones, until a global number of nMaxClusters is reached. *)
		bSingleSplitSteps	:	BOOL;	(* If true, the global optimization is always run after a single cluster has been split. If false, several clusters are split within the same step before applying the global optimization. Applying the global optimization less often is faster, but can lead to less optimal results, especially having 2 nearby clusters that could be represented by 1. *)
		hrPrev	:	HRESULT;	(* HRESULT indicating the result of previous operations (If SUCCEEDED(hrPrev) equals false, no operation is executed.) *)
	END_VAR

END_FUNCTION

// Functions/Machine Learning/F_VN_CreateLbgModelExp

	{attribute 'TcIecLibraryType'}
	{attribute 'external_name' := 'F_VN_CreateLbgModelExp_GUID_7D80325A_5FE2_204A_5847_DCDBD3907200'}
	(* Create a LBG model of the specified type. The initial reference count is set to one if a new model is created and kept, otherwise. Models of this type neither support on-line training (sample by sample) nor retraining. (expert function) *)
	FUNCTION F_VN_CreateLbgModelExp : HRESULT
	VAR_INPUT
		ipMlModel	:	REFERENCE TO ITcVnMlModel;	(* Returns the created model (Non-zero interface pointers are reused.) *)
		eLbgType	:	ETcVnPrototypeClusterer;	(* LBG model type *)
		nMaxClusters	:	UDINT;	(* Maximum number of clusters *)
		fMaxClusterRadius	:	LREAL;	(* Maximum allowed radius (L2 norm) of a single cluster, i.e. clusters with a higher radius will be split into smaller ones, until a global number of nMaxClusters is reached. *)
		bSingleSplitSteps	:	BOOL;	(* If true, the global optimization is always run after a single cluster has been split. If false, several clusters are split within the same step before applying the global optimization. Applying the global optimization less often is faster, but can lead to less optimal results, especially having 2 nearby clusters that could be represented by 1. *)
		bDoublePrecision	:	BOOL;	(* If true, the model is generated with double precision (LREAL) instead of single precision (REAL). (default: FALSE) *)
		nMaxIterations	:	UDINT;	(* Maximum number of iterations (triggers the usage of the default value of 10 if it equals 0) *)
		fEpsilon	:	LREAL;	(* Maximum allowed difference of the error between two successive iterations (triggers the usage of the default value of 0.001 if it equals 0) *)
		hrPrev	:	HRESULT;	(* HRESULT indicating the result of previous operations (If SUCCEEDED(hrPrev) equals false, no operation is executed.) *)
	END_VAR

END_FUNCTION

// Functions/Machine Learning/F_VN_CreateLdaTransform

	{attribute 'TcIecLibraryType'}
	{attribute 'external_name' := 'F_VN_CreateLdaTransform_GUID_BFEE6E72_265C_2874_673C_367B017B49AA'}
	(* Create an LDA-based feature transform from the provided data. The number of samples must be >= the number of features and the number of classes must be >= 2. The initial reference count is set to one if a new model is created and kept, otherwise. *)
	FUNCTION F_VN_CreateLdaTransform : HRESULT
	VAR_INPUT
		ipMlModel	:	REFERENCE TO ITcVnMlModel;	(* Returns the created feature transform (Non-zero interface pointers are reused.) *)
		ipSamples	:	ITcUnknown;	(* Container holding a batch of input samples (ContainerType_Vector_Vector_REAL or ContainerType_Vector_Vector_LREAL) *)
		ipClasses	:	ITcVnContainer;	(* Class labels corresponding to the input samples (ContainerType_Vector_DINT) *)
		hrPrev	:	HRESULT;	(* HRESULT indicating the result of previous operations (If SUCCEEDED(hrPrev) equals false, no operation is executed.) *)
	END_VAR

END_FUNCTION

// Functions/Machine Learning/F_VN_CreateLdaTransformViaComponentNum

	{attribute 'TcIecLibraryType'}
	{attribute 'external_name' := 'F_VN_CreateLdaTransformViaComponentNum_GUID_9BEA4391_283A_253A_73D7_A94E3C32FB17'}
	(* Create an LDA-based feature transform from the provided data where the number of components to be used is predefined. The number of samples must be >= the number of features and the number of classes must be >= 2. The initial reference count is set to one if a new model is created and kept, otherwise. (expert function) *)
	FUNCTION F_VN_CreateLdaTransformViaComponentNum : HRESULT
	VAR_INPUT
		ipMlModel	:	REFERENCE TO ITcVnMlModel;	(* Returns the created feature transform (Non-zero interface pointers are reused.) *)
		ipSamples	:	ITcUnknown;	(* Container holding a batch of input samples (ContainerType_Vector_Vector_REAL or ContainerType_Vector_Vector_LREAL) *)
		ipClasses	:	ITcVnContainer;	(* Class labels corresponding to the input samples (ContainerType_Vector_DINT) *)
		nComponentNum	:	UDINT;	(* Number of components (nComponentNum must be smaller than the number of classes. A value of 0 results in the automatic computation of the maximum number of components.) *)
		hrPrev	:	HRESULT;	(* HRESULT indicating the result of previous operations (If SUCCEEDED(hrPrev) equals false, no operation is executed.) *)
	END_VAR

END_FUNCTION

// Functions/Machine Learning/F_VN_CreateNbcModel

	{attribute 'TcIecLibraryType'}
	{attribute 'external_name' := 'F_VN_CreateNbcModel_GUID_DA02C3CE_3432_20F0_76B8_8F9342393153'}
	(* Create a normal Bayes classifier of the specified type. The initial reference count is set to one if a new model is created and kept, otherwise. In order to train normal Bayes classifiers, a sufficiently high number of samples is required for each class. It depends on the number of features and the distribution of the data. Hence, it needs to be tested for each application. Models of this type do not support on-line training (sample by sample). For the retraining of such classifier models, the set of presented classes must be identical to the previous learning steps. Otherwise, an exception is raised. *)
	FUNCTION F_VN_CreateNbcModel : HRESULT
	VAR_INPUT
		ipMlModel	:	REFERENCE TO ITcVnMlModel;	(* Returns the created model (Non-zero interface pointers are reused.) *)
		eNbcType	:	ETcVnNbc;	(* Normal Bayes classifier type *)
		hrPrev	:	HRESULT;	(* HRESULT indicating the result of previous operations (If SUCCEEDED(hrPrev) equals false, no operation is executed.) *)
	END_VAR

END_FUNCTION

// Functions/Machine Learning/F_VN_CreatePcaTransform

	{attribute 'TcIecLibraryType'}
	{attribute 'external_name' := 'F_VN_CreatePcaTransform_GUID_DA24C08E_FFC7_2FDD_40DC_07CC6EFE8395'}
	(* Create a PCA-based feature transform from the provided data. The maximum number of principal components that can be computed equals the minimum of the number of samples and the number of features. The initial reference count is set to one if a new model is created and kept, otherwise. *)
	FUNCTION F_VN_CreatePcaTransform : HRESULT
	VAR_INPUT
		ipMlModel	:	REFERENCE TO ITcVnMlModel;	(* Returns the created feature transform (Non-zero interface pointers are reused.) *)
		ipSamples	:	ITcUnknown;	(* Container holding a batch of input samples (ContainerType_Vector_Vector_REAL or ContainerType_Vector_Vector_LREAL) *)
		hrPrev	:	HRESULT;	(* HRESULT indicating the result of previous operations (If SUCCEEDED(hrPrev) equals false, no operation is executed.) *)
	END_VAR

END_FUNCTION

// Functions/Machine Learning/F_VN_CreatePcaTransformViaComponentNum

	{attribute 'TcIecLibraryType'}
	{attribute 'external_name' := 'F_VN_CreatePcaTransformViaComponentNum_GUID_28104B27_51EA_20F4_57BD_7EF798538D8F'}
	(* Create a PCA-based feature transform from the provided data where the number of prinicpal components to be used is predefined. The maximum number of principal components that can be computed equals the minimum of the number of samples and the number of features. The initial reference count is set to one if a new model is created and kept, otherwise. (expert function) *)
	FUNCTION F_VN_CreatePcaTransformViaComponentNum : HRESULT
	VAR_INPUT
		ipMlModel	:	REFERENCE TO ITcVnMlModel;	(* Returns the created feature transform (Non-zero interface pointers are reused.) *)
		ipSamples	:	ITcUnknown;	(* Container holding a batch of input samples (ContainerType_Vector_Vector_REAL or ContainerType_Vector_Vector_LREAL) *)
		nComponentNum	:	UDINT;	(* Number of principal components (A value of 0 results in the automatic computation of the maximum number of components.) *)
		hrPrev	:	HRESULT;	(* HRESULT indicating the result of previous operations (If SUCCEEDED(hrPrev) equals false, no operation is executed.) *)
	END_VAR

END_FUNCTION

// Functions/Machine Learning/F_VN_CreatePcaTransformViaVariance

	{attribute 'TcIecLibraryType'}
	{attribute 'external_name' := 'F_VN_CreatePcaTransformViaVariance_GUID_1D00BCB6_0F8E_2453_7A66_86E326231A6F'}
	(* Create a PCA-based feature transform from the provided data based on a given fraction of variance to be retained. The maximum number of principal components that can be computed equals the minimum of the number of samples and the number of features. The initial reference count is set to one if a new model is created and kept, otherwise. (expert function) *)
	FUNCTION F_VN_CreatePcaTransformViaVariance : HRESULT
	VAR_INPUT
		ipMlModel	:	REFERENCE TO ITcVnMlModel;	(* Returns the created feature transform (Non-zero interface pointers are reused.) *)
		ipSamples	:	ITcUnknown;	(* Container holding a batch of input samples (ContainerType_Vector_Vector_REAL or ContainerType_Vector_Vector_LREAL) *)
		fRetainedVariance	:	LREAL;	(* Fraction of variance that is to be retained by the PCA (A value of 1.0 signifies 100%.) *)
		hrPrev	:	HRESULT;	(* HRESULT indicating the result of previous operations (If SUCCEEDED(hrPrev) equals false, no operation is executed.) *)
	END_VAR

END_FUNCTION

// Functions/Machine Learning/F_VN_CreateRTreesModel

	{attribute 'TcIecLibraryType'}
	{attribute 'external_name' := 'F_VN_CreateRTreesModel_GUID_5E8D1899_6C3A_2CDF_5A6E_02E699F01A9E'}
	(* Create a random trees model of the specified type. The initial reference count is set to one if a new model is created and kept, otherwise. Models of this type neither support on-line training (sample by sample) nor retraining. Predictions can only be scalar. *)
	FUNCTION F_VN_CreateRTreesModel : HRESULT
	VAR_INPUT
		ipMlModel	:	REFERENCE TO ITcVnMlModel;	(* Returns the created model (Non-zero interface pointers are reused.) *)
		eRTreesType	:	ETcVnRTrees;	(* Random trees model type *)
		hrPrev	:	HRESULT;	(* HRESULT indicating the result of previous operations (If SUCCEEDED(hrPrev) equals false, no operation is executed.) *)
	END_VAR

END_FUNCTION

// Functions/Machine Learning/F_VN_CreateRTreesModelExp

	{attribute 'TcIecLibraryType'}
	{attribute 'external_name' := 'F_VN_CreateRTreesModelExp_GUID_B4393A32_59CB_20BD_6E6F_3D9FC67F97F8'}
	(* Create a random trees model of the specified type. The initial reference count is set to one if a new model is created and kept, otherwise. Models of this type neither support on-line training (sample by sample) nor retraining. Predictions can only be scalar. (expert function) *)
	FUNCTION F_VN_CreateRTreesModelExp : HRESULT
	VAR_INPUT
		ipMlModel	:	REFERENCE TO ITcVnMlModel;	(* Returns the created model (Non-zero interface pointers are reused.) *)
		eRTreesType	:	ETcVnRTrees;	(* Random trees model type *)
		nMaxDepth	:	UDINT;	(* Maximum tree depth (default: 5) *)
		nMinSamples	:	UDINT;	(* Minimum number of samples within a node required for splitting (default: 10) *)
		nActiveVariables	:	UDINT;	(* Number of variables considered for splitting (0 means sqrt(total number of variables); default: 0) *)
		nMaxIterations	:	UDINT;	(* Maximum number of iterations (disabled if it equals 0 and fEpsilon is different from 0.0; triggers the usage of the default value of 50 if nMaxIterations and fEpsilon equal 0) *)
		fEpsilon	:	LREAL;	(* Maximum allowed difference of the error between two successive iterations (disabled if it equals 0.0 and nMaxIterations is different from 0; triggers the usage of the default value of 0.1 if nMaxIterations and fEpsilon equal 0) *)
		hrPrev	:	HRESULT;	(* HRESULT indicating the result of previous operations (If SUCCEEDED(hrPrev) equals false, no operation is executed.) *)
	END_VAR

END_FUNCTION

// Functions/Machine Learning/F_VN_CreateRTreesModelExp2

	{attribute 'TcIecLibraryType'}
	{attribute 'external_name' := 'F_VN_CreateRTreesModelExp2_GUID_CB2A007E_1A54_217F_7384_3FD84203AD44'}
	(* Create a random trees model of the specified type. The initial reference count is set to one if a new model is created and kept, otherwise. Models of this type neither support on-line training (sample by sample) nor retraining. Predictions can only be scalar. (expert function) *)
	FUNCTION F_VN_CreateRTreesModelExp2 : HRESULT
	VAR_INPUT
		ipMlModel	:	REFERENCE TO ITcVnMlModel;	(* Returns the created model (Non-zero interface pointers are reused.) *)
		eRTreesType	:	ETcVnRTrees;	(* Random trees model type *)
		nMaxDepth	:	UDINT;	(* Maximum tree depth (default: 5) *)
		nMinSamples	:	UDINT;	(* Minimum number of samples within a node required for splitting (default: 10) *)
		nActiveVariables	:	UDINT;	(* Number of variables considered for splitting (0 means sqrt(total number of variables); default: 0) *)
		nMaxIterations	:	UDINT;	(* Maximum number of iterations (disabled if it equals 0 and fEpsilon is different from 0.0; triggers the usage of the default value of 50 if nMaxIterations and fEpsilon equal 0) *)
		fEpsilon	:	LREAL;	(* Maximum allowed difference of the error between two successive iterations (disabled if it equals 0.0 and nMaxIterations is different from 0; triggers the usage of the default value of 0.1 if nMaxIterations and fEpsilon equal 0) *)
		fRegressionAccuracy	:	REAL;	(* Termination criterion for regressors (only for regressors; set to default if not allowed; default: 0.0) *)
		ipClassPriors	:	ITcVnContainer;	(* Class priors (ContainerType_Vector_REAL or ContainerType_Vector_LREAL; only for classifiers; optional, set to 0 if not required or not allowed; default: 0) *)
		hrPrev	:	HRESULT;	(* HRESULT indicating the result of previous operations (If SUCCEEDED(hrPrev) equals false, no operation is executed.) *)
	END_VAR

END_FUNCTION

// Functions/Machine Learning/F_VN_CreateStaModel

	{attribute 'TcIecLibraryType'}
	{attribute 'external_name' := 'F_VN_CreateStaModel_GUID_66F6A4E1_5161_2538_5E15_959ACE2242A0'}
	(* Create a Simplified TopoART neural network of the specified type. The initial reference count is set to one if a new model is created and kept, otherwise. Models of this type support on-line training (sample by sample), retraining, as well as scalar and vectorial predictions. It requires all input except class labels (i.e., samples and training outputs/predictions) to lie in the interval [0.0, 1.0]. The predictions of regressors need to be rescaled from the interval [0.0, 1.0] to their respective value range before usage. Depending on the parameter settings and the number of available training samples, repeated training with the same data may improve the results. Like other neural networks based on the Adaptive Resonance Theory (ART), Simplified TopoART neural networks are not prone to catastrophic inference and patricularly well-suited to incremental learning tasks. *)
	FUNCTION F_VN_CreateStaModel : HRESULT
	VAR_INPUT
		ipMlModel	:	REFERENCE TO ITcVnMlModel;	(* Returns the created model (Non-zero interface pointers are reused.) *)
		eStaType	:	ETcVnSta;	(* Simpified TopoART model type *)
		fRho	:	LREAL;	(* Vigilance parameter (controls the number of neurons that are inserted and the maximum size of the formed categories; valid range: [0.0, 1.0]; suggested range: [0.8, 1.0)) *)
		hrPrev	:	HRESULT;	(* HRESULT indicating the result of previous operations (If SUCCEEDED(hrPrev) equals false, no operation is executed.) *)
	END_VAR

END_FUNCTION

// Functions/Machine Learning/F_VN_CreateStaModelExp

	{attribute 'TcIecLibraryType'}
	{attribute 'external_name' := 'F_VN_CreateStaModelExp_GUID_085A0D33_A299_2BF8_4BAF_C8D386BECA2F'}
	(* Create a Simplified TopoART neural network of the specified type. The initial reference count is set to one if a new model is created and kept, otherwise. Models of this type support on-line training (sample by sample), retraining, as well as scalar and vectorial predictions. It requires all input except class labels (i.e., samples and training outputs/predictions) to lie in the interval [0.0, 1.0]. The predictions of regressors need to be rescaled from the interval [0.0, 1.0] to their respective value range before usage. Depending on the parameter settings and the number of available training samples, repeated training with the same data may improve the results. Like other neural networks based on the Adaptive Resonance Theory (ART), Simplified TopoART neural networks are not prone to catastrophic inference and patricularly well-suited to incremental learning tasks. (expert function) *)
	FUNCTION F_VN_CreateStaModelExp : HRESULT
	VAR_INPUT
		ipMlModel	:	REFERENCE TO ITcVnMlModel;	(* Returns the created model (Non-zero interface pointers are reused.) *)
		eStaType	:	ETcVnSta;	(* Simpified TopoART model type *)
		fRho	:	LREAL;	(* Vigilance parameter (controls the number of neurons that are inserted and the maximum size of the formed categories; valid range: [0.0, 1.0]; suggested range: [0.8, 1.0)) *)
		nNu	:	UDINT;	(* Number of neurons used for classification and prediction (must be larger than or equal to 1; suggested range: [1, 10); default: 3) *)
		bDoublePrecision	:	BOOL;	(* If true, the model is generated with double precision (LREAL) instead of single precision (REAL). (default: FALSE) *)
		hrPrev	:	HRESULT;	(* HRESULT indicating the result of previous operations (If SUCCEEDED(hrPrev) equals false, no operation is executed.) *)
	END_VAR

END_FUNCTION

// Functions/Machine Learning/F_VN_CreateStaModelExp2

	{attribute 'TcIecLibraryType'}
	{attribute 'external_name' := 'F_VN_CreateStaModelExp2_GUID_B4C9EC77_862D_2DD5_5390_92D4C6B86CC8'}
	(* Create a Simplified TopoART neural network of the specified type. The initial reference count is set to one if a new model is created and kept, otherwise. Models of this type support on-line training (sample by sample), retraining, as well as scalar and vectorial predictions. It requires all input except class labels (i.e., samples and training outputs/predictions) to lie in the interval [0.0, 1.0]. The predictions of regressors need to be rescaled from the interval [0.0, 1.0] to their respective value range before usage. Depending on the parameter settings and the number of available training samples, repeated training with the same data may improve the results. Like other neural networks based on the Adaptive Resonance Theory (ART), Simplified TopoART neural networks are not prone to catastrophic inference and patricularly well-suited to incremental learning tasks. (additional expert function providing parameters for fine-tuning and noise reduction) *)
	FUNCTION F_VN_CreateStaModelExp2 : HRESULT
	VAR_INPUT
		ipMlModel	:	REFERENCE TO ITcVnMlModel;	(* Returns the created model (Non-zero interface pointers are reused.) *)
		eStaType	:	ETcVnSta;	(* Simpified TopoART model type *)
		fRho	:	LREAL;	(* Vigilance parameter (controls the number of neurons that are inserted and the maximum size of the formed categories; valid range: [0.0, 1.0]; suggested range: [0.8, 1.0)) *)
		nNu	:	UDINT;	(* Number of neurons used for classification and prediction (must be larger than or equal to 1; suggested range: [1, 10); default: 3) *)
		bDoublePrecision	:	BOOL;	(* If true, the model is generated with double precision (LREAL) instead of single precision (REAL). (default: FALSE) *)
		fBetaSbm	:	LREAL;	(* Learning rate of the second best-matching neuron (learning the second best-matching neuron keeps related categories closer together and might improve the results but may require a higher number of neurons and training runs; a value of 0.0 disables learning of the second best-matching neuron; valid range: [0.0, 1.0]; suggested range: [0.0, 0.5]); default: 0.0 *)
		nPhi	:	UDINT;	(* Number of samples a neuron must have learnt to become permanent (required for noise reduction; works in conjunction with nTau; must be larger than or equal to 1; higher values intensify noise reduction; a value of 1 disables removal of neuron candidates; default: 1) *)
		nTau	:	UDINT;	(* Number of learning steps after which node removal is performed (required for noise reduction; works in conjunction with nPhi; must be large enough to allow neuron candidates representing non-noise samples to become the best-matching neuron at least nPhi times before node removal; default: 100) *)
		hrPrev	:	HRESULT;	(* HRESULT indicating the result of previous operations (If SUCCEEDED(hrPrev) equals false, no operation is executed.) *)
	END_VAR

END_FUNCTION

// Functions/Machine Learning/F_VN_CreateSvmModel

	{attribute 'TcIecLibraryType'}
	{attribute 'external_name' := 'F_VN_CreateSvmModel_GUID_0E9B46AA_E9FD_244C_7078_B9DB23BF7170'}
	(* Create an SVM model of the specified type. The initial reference count is set to one if a new model is created and kept, otherwise. Models of this type neither support on-line training (sample by sample) nor retraining. Predictions can only be scalar. *)
	FUNCTION F_VN_CreateSvmModel : HRESULT
	VAR_INPUT
		ipMlModel	:	REFERENCE TO ITcVnMlModel;	(* Returns the created model (Non-zero interface pointers are reused.) *)
		eSvmType	:	ETcVnSvm;	(* SVM model type *)
		fC	:	LREAL;	(* Parameter C (required for TCVN_SVM_C_CLASSIFIER, TCVN_SVM_EPS_REGRESSOR, and TCVN_SVM_NU_REGRESSOR; ignored otherwise) *)
		fNu	:	LREAL;	(* Parameter nu (required for TCVN_SVM_NU_CLASSIFIER, TCVN_SVM_NOVELTY_DETECTOR, and TCVN_SVM_NU_REGRESSOR; ignored otherwise) *)
		fP	:	LREAL;	(* Parameter p (required for TCVN_SVM_EPS_REGRESSOR; ignored otherwise) *)
		eKernelType	:	ETcVnSvmKernelType;	(* Kernel type *)
		fGamma	:	LREAL;	(* Parameter gamma (used by polynomial, RBF, sigmoid, and chi-squared kernels; ignored otherwise) *)
		fCoef0	:	LREAL;	(* parameter coef0 (used by polynomial and sigmoid kernels; ignored otherwise) *)
		fDegree	:	LREAL;	(* Degree (used by polynomial kernels; ignored otherwise) *)
		hrPrev	:	HRESULT;	(* HRESULT indicating the result of previous operations (If SUCCEEDED(hrPrev) equals false, no operation is executed.) *)
	END_VAR

END_FUNCTION

// Functions/Machine Learning/F_VN_CreateSvmModelExp

	{attribute 'TcIecLibraryType'}
	{attribute 'external_name' := 'F_VN_CreateSvmModelExp_GUID_038EDCA5_BA03_2CC3_41B7_ACD066032535'}
	(* Create an SVM model of the specified type. The initial reference count is set to one if a new model is created and kept, otherwise. Models of this type neither support on-line training (sample by sample) nor retraining. Predictions can only be scalar. (expert function) *)
	FUNCTION F_VN_CreateSvmModelExp : HRESULT
	VAR_INPUT
		ipMlModel	:	REFERENCE TO ITcVnMlModel;	(* Returns the created model (Non-zero interface pointers are reused.) *)
		eSvmType	:	ETcVnSvm;	(* SVM model type *)
		fC	:	LREAL;	(* Parameter C (required for TCVN_SVM_C_CLASSIFIER, TCVN_SVM_EPS_REGRESSOR, and TCVN_SVM_NU_REGRESSOR; ignored otherwise) *)
		fNu	:	LREAL;	(* Parameter nu (required for TCVN_SVM_NU_CLASSIFIER, TCVN_SVM_NOVELTY_DETECTOR, and TCVN_SVM_NU_REGRESSOR; ignored otherwise) *)
		fP	:	LREAL;	(* Parameter p (required for TCVN_SVM_EPS_REGRESSOR; ignored otherwise) *)
		eKernelType	:	ETcVnSvmKernelType;	(* Kernel type *)
		fGamma	:	LREAL;	(* Parameter gamma (used by polynomial, RBF, sigmoid, and chi-squared kernels; ignored otherwise) *)
		fCoef0	:	LREAL;	(* Parameter coef0 (used by polynomial and sigmoid kernels; ignored otherwise) *)
		fDegree	:	LREAL;	(* Degree (used by polynomial kernels; ignored otherwise) *)
		nMaxIterations	:	UDINT;	(* Maximum number of iterations (disabled if it equals 0 and fEpsilon is different from 0.0; triggers the usage of the default value of 100000 if nMaxIterations and fEpsilon equal 0) *)
		fEpsilon	:	LREAL;	(* Maximum allowed difference of the error between two successive iterations (disabled if it equals 0.0 and nMaxIterations is different from 0; triggers the usage of the default value of 0.00001 if nMaxIterations and fEpsilon equal 0) *)
		hrPrev	:	HRESULT;	(* HRESULT indicating the result of previous operations (If SUCCEEDED(hrPrev) equals false, no operation is executed.) *)
	END_VAR

END_FUNCTION

// Functions/Machine Learning/F_VN_CreateSvmModelExp2

	{attribute 'TcIecLibraryType'}
	{attribute 'external_name' := 'F_VN_CreateSvmModelExp2_GUID_0746A115_4AF6_2638_52C1_AF37A6B8EC60'}
	(* Create an SVM model of the specified type. The initial reference count is set to one if a new model is created and kept, otherwise. Models of this type neither support on-line training (sample by sample) nor retraining. Predictions can only be scalar. (additional expert function for C support vector classifiers) *)
	FUNCTION F_VN_CreateSvmModelExp2 : HRESULT
	VAR_INPUT
		ipMlModel	:	REFERENCE TO ITcVnMlModel;	(* Returns the created model (Non-zero interface pointers are reused.) *)
		eSvmType	:	ETcVnSvm;	(* SVM model type *)
		fC	:	LREAL;	(* Parameter C (required for TCVN_SVM_C_CLASSIFIER, TCVN_SVM_EPS_REGRESSOR, and TCVN_SVM_NU_REGRESSOR; ignored otherwise) *)
		fNu	:	LREAL;	(* Parameter nu (required for TCVN_SVM_NU_CLASSIFIER, TCVN_SVM_NOVELTY_DETECTOR, and TCVN_SVM_NU_REGRESSOR; ignored otherwise) *)
		fP	:	LREAL;	(* Parameter p (required for TCVN_SVM_EPS_REGRESSOR; ignored otherwise) *)
		eKernelType	:	ETcVnSvmKernelType;	(* Kernel type *)
		fGamma	:	LREAL;	(* Parameter gamma (used by polynomial, RBF, sigmoid, and chi-squared kernels; ignored otherwise) *)
		fCoef0	:	LREAL;	(* Parameter coef0 (used by polynomial and sigmoid kernels; ignored otherwise) *)
		fDegree	:	LREAL;	(* Degree (used by polynomial kernels; ignored otherwise) *)
		nMaxIterations	:	UDINT;	(* Maximum number of iterations (disabled if it equals 0 and fEpsilon is different from 0.0; triggers the usage of the default value of 100000 if nMaxIterations and fEpsilon equal 0) *)
		fEpsilon	:	LREAL;	(* Maximum allowed difference of the error between two successive iterations (disabled if it equals 0.0 and nMaxIterations is different from 0; triggers the usage of the default value of 0.00001 if nMaxIterations and fEpsilon equal 0) *)
		ipClassWeights	:	ITcVnContainer;	(* Class weights (ContainerType_Vector_REAL or ContainerType_Vector_LREAL; only valid if eSvmType equals TCVN_SVM_C_CLASSIFIER; optional, set to 0 if not required or not allowed; default: 0) *)
		hrPrev	:	HRESULT;	(* HRESULT indicating the result of previous operations (If SUCCEEDED(hrPrev) equals false, no operation is executed.) *)
	END_VAR

END_FUNCTION

// Functions/Machine Learning/F_VN_CreateSvmSgdClassifier

	{attribute 'TcIecLibraryType'}
	{attribute 'external_name' := 'F_VN_CreateSvmSgdClassifier_GUID_A17D7728_A7F2_2008_690B_C59E5F8E21BB'}
	(* Create a linear SVM classifier using stochastic gradient descent for training. The initial reference count is set to one if a new model is created and kept, otherwise. This SVM classifier is only applicable to binary classification problems. It learns a separating hyperplane between a class with label -1 and a class with label 1. These class labels are predefined. For training, any positive class labels are mapped to 1 and any negative class labels are mapped to -1. Models of this type neither support on-line training (sample by sample) nor retraining. *)
	FUNCTION F_VN_CreateSvmSgdClassifier : HRESULT
	VAR_INPUT
		ipMlModel	:	REFERENCE TO ITcVnMlModel;	(* Returns the created model (Non-zero interface pointers are reused.) *)
		hrPrev	:	HRESULT;	(* HRESULT indicating the result of previous operations (If SUCCEEDED(hrPrev) equals false, no operation is executed.) *)
	END_VAR

END_FUNCTION

// Functions/Machine Learning/F_VN_CreateSvmSgdClassifierExp

	{attribute 'TcIecLibraryType'}
	{attribute 'external_name' := 'F_VN_CreateSvmSgdClassifierExp_GUID_5DE27E7E_DC42_23D2_4668_7DD1EE684C9B'}
	(* Create a linear SVM classifier using stochastic gradient descent for training. The initial reference count is set to one if a new model is created and kept, otherwise. This SVM classifier is only applicable to binary classification problems. It learns a separating hyperplane between a class with label -1 and a class with label 1. These class labels are predefined. For training, any positive class labels are mapped to 1 and any negative class labels are mapped to -1. Models of this type neither support on-line training (sample by sample) nor retraining. (expert function) *)
	FUNCTION F_VN_CreateSvmSgdClassifierExp : HRESULT
	VAR_INPUT
		ipMlModel	:	REFERENCE TO ITcVnMlModel;	(* Returns the created model (Non-zero interface pointers are reused.) *)
		eType	:	ETcVnSvmSgdClassifierType;	(* Learning algorithm type (default: TCVN_SSCT_ASGD) *)
		eMarginType	:	ETcVnSvmSgdClassifierMarginType;	(* Margin type (default: TCVN_SSCMT_SOFT_MARGIN) *)
		fMarginRegularization	:	REAL;	(* Margin regularization parameter (default: 0.00001) *)
		fInitialStepSize	:	REAL;	(* Initial step size (default: 0.05) *)
		fStepDecreasingPower	:	REAL;	(* Power parameter (default: 0.75) *)
		nMaxIterations	:	UDINT;	(* Maximum number of iterations (disabled if it equals 0 and fEpsilon is different from 0.0; triggers the usage of the default value of 100000 if nMaxIterations and fEpsilon equal 0) *)
		fEpsilon	:	LREAL;	(* Maximum allowed difference of the error between two successive iterations (disabled if it equals 0.0 and nMaxIterations is different from 0; triggers the usage of the default value of 0.00001 if nMaxIterations and fEpsilon equal 0) *)
		hrPrev	:	HRESULT;	(* HRESULT indicating the result of previous operations (If SUCCEEDED(hrPrev) equals false, no operation is executed.) *)
	END_VAR

END_FUNCTION

// Functions/Machine Learning/F_VN_FeatureTransform

	{attribute 'TcIecLibraryType'}
	{attribute 'external_name' := 'F_VN_FeatureTransform_GUID_AE94F9F9_DCE5_2E54_6414_1C537994E59A'}
	(* Apply a feature transform to one or more sample(s). *)
	FUNCTION F_VN_FeatureTransform : HRESULT
	VAR_INPUT
		ipFeatureTransform	:	ITcVnMlModel;	(* Feature transform instance to be used *)
		ipSamples	:	ITcUnknown;	(* Container holding one or more of input sample(s) (ContainerType_Vector_REAL, ContainerType_Vector_LREAL, ContainerType_Vector_Vector_REAL, or ContainerType_Vector_Vector_LREAL) *)
		pipTransformed	:	POINTER TO ITcUnknown;	(* Returns the transformed sample(s) using the same type like ipSamples *)
		hrPrev	:	HRESULT;	(* HRESULT indicating the result of previous operations (If SUCCEEDED(hrPrev) equals false, no operation is executed.) *)
	END_VAR

END_FUNCTION

// Functions/Machine Learning/F_VN_GetBatchClusters

	{attribute 'TcIecLibraryType'}
	{attribute 'external_name' := 'F_VN_GetBatchClusters_GUID_3A1D7A9A_EF4E_2678_5016_66C5AD05593C'}
	(* Get the IDs of the best-matching clusters of a batch of samples. *)
	FUNCTION F_VN_GetBatchClusters : HRESULT
	VAR_INPUT
		ipClusterer	:	ITcVnMlModel;	(* Clusterer to be used *)
		ipSamples	:	ITcUnknown;	(* Container holding a batch of input samples (ContainerType_Vector_Vector_REAL or ContainerType_Vector_Vector_LREAL) *)
		ipClusters	:	REFERENCE TO ITcVnContainer;	(* Returns the cluster IDs (ContainerType_Vector_DINT) *)
		hrPrev	:	HRESULT;	(* HRESULT indicating the result of previous operations (If SUCCEEDED(hrPrev) equals false, no operation is executed.) *)
	END_VAR

END_FUNCTION

// Functions/Machine Learning/F_VN_GetBatchClustersExp

	{attribute 'TcIecLibraryType'}
	{attribute 'external_name' := 'F_VN_GetBatchClustersExp_GUID_82B4EDF3_30DD_212D_6B2A_DD339AA48928'}
	(* Get the IDs of the best-matching clusters of a batch of samples. *)
	FUNCTION F_VN_GetBatchClustersExp : HRESULT
	VAR_INPUT
		ipClusterer	:	ITcVnMlModel;	(* Clusterer to be used *)
		ipSamples	:	ITcUnknown;	(* Container holding a batch of input samples (ContainerType_Vector_Vector_REAL or ContainerType_Vector_Vector_LREAL) *)
		ipClusters	:	REFERENCE TO ITcVnContainer;	(* Returns the cluster IDs (ContainerType_Vector_DINT) *)
		ipNovelties	:	REFERENCE TO ITcVnContainer;	(* Returns the degree of novelty (0.0 if a sample is completely known; > 0.0 otherwise) of each sample (ContainerType_Vector_REAL; optional, set to 0 if not required) *)
		hrPrev	:	HRESULT;	(* HRESULT indicating the result of previous operations (If SUCCEEDED(hrPrev) equals false, no operation is executed.) *)
	END_VAR

END_FUNCTION

// Functions/Machine Learning/F_VN_GetBatchNovelties

	{attribute 'TcIecLibraryType'}
	{attribute 'external_name' := 'F_VN_GetBatchNovelties_GUID_14A8FD94_D495_2B7B_5C7B_B2C132CF0190'}
	(* Get the degree of novelty of multiple samples. *)
	FUNCTION F_VN_GetBatchNovelties : HRESULT
	VAR_INPUT
		ipNoveltyDetector	:	ITcVnMlModel;	(* Novelty detector to be used *)
		ipSamples	:	ITcUnknown;	(* Container holding a batch of input samples (ContainerType_Vector_Vector_REAL or ContainerType_Vector_Vector_LREAL) *)
		ipNovelties	:	REFERENCE TO ITcVnContainer;	(* Returns the degree of novelty (0.0 if a sample is completely known; > 0.0 otherwise) of each sample (ContainerType_Vector_REAL) *)
		hrPrev	:	HRESULT;	(* HRESULT indicating the result of previous operations (If SUCCEEDED(hrPrev) equals false, no operation is executed.) *)
	END_VAR

END_FUNCTION

// Functions/Machine Learning/F_VN_GetClusterCenter

	{attribute 'TcIecLibraryType'}
	{attribute 'external_name' := 'F_VN_GetClusterCenter_GUID_671FEDB4_4237_2A4A_544A_86F4900FEADE'}
	(* Get the center of a cluster. *)
	FUNCTION F_VN_GetClusterCenter : HRESULT
	VAR_INPUT
		ipClusterer	:	ITcVnMlModel;	(* Clusterer to be used *)
		nCluster	:	DINT;	(* Cluster ID of the cluster the center of which is requested *)
		ipCenter	:	REFERENCE TO ITcVnContainer;	(* Returns the cluster center (ContainerType_Vector_REAL or ContainerType_Vector_LREAL depending on the floating point type internally used by the clusterer) *)
		hrPrev	:	HRESULT;	(* HRESULT indicating the result of previous operations (If SUCCEEDED(hrPrev) equals false, no operation is executed.) *)
	END_VAR

END_FUNCTION

// Functions/Machine Learning/F_VN_GetClusterNum

	{attribute 'TcIecLibraryType'}
	{attribute 'external_name' := 'F_VN_GetClusterNum_GUID_3C1C2FBE_3CBA_21B5_765A_28AF0ECDBB5D'}
	(* Get the number of clusters used by this clusterer. *)
	FUNCTION F_VN_GetClusterNum : HRESULT
	VAR_INPUT
		ipClusterer	:	ITcVnMlModel;	(* Clusterer to be used *)
	END_VAR
	VAR_IN_OUT
		nClusterNum	:	ULINT;	(* Returns the number of clusters *)
	END_VAR
	VAR_INPUT
		hrPrev	:	HRESULT;	(* HRESULT indicating the result of previous operations (If SUCCEEDED(hrPrev) equals false, no operation is executed.) *)
	END_VAR

END_FUNCTION

// Functions/Machine Learning/F_VN_GetFeatureScales

	{attribute 'TcIecLibraryType'}
	{attribute 'external_name' := 'F_VN_GetFeatureScales_GUID_96A5CB44_57E6_2A7D_56CA_F7ABA73E8752'}
	(* Calculate the scaling parameters for each feature in the input samples based on the scaling type. *)
	FUNCTION F_VN_GetFeatureScales : HRESULT
	VAR_INPUT
		ipSamples	:	ITcVnContainer;	(* Container holding input sample(s) (ContainerType_Vector_REAL, ContainerType_Vector_LREAL, ContainerType_Vector_Vector_REAL or ContainerType_Vector_Vector_LREAL) *)
		ipScales	:	REFERENCE TO ITcVnContainer;	(* Returns a container with the scaling parameters for each feature (Vector_REAL or Vector_LREAL depending on the type of ipSamples). *)
		eFeatureScalingType	:	ETcVnFeatureScalingType;	(* Feature scaling type *)
		hrPrev	:	HRESULT;	(* HRESULT indicating the result of previous operations (If SUCCEEDED(hrPrev) equals false, no operation is executed.) *)
	END_VAR

END_FUNCTION

// Functions/Machine Learning/F_VN_GetSampleCluster

	{attribute 'TcIecLibraryType'}
	{attribute 'external_name' := 'F_VN_GetSampleCluster_GUID_5A615556_C62E_23E0_490A_36F4F321DCCB'}
	(* Get the ID of the best-matching cluster of a single sample. *)
	FUNCTION F_VN_GetSampleCluster : HRESULT
	VAR_INPUT
		ipClusterer	:	ITcVnMlModel;	(* Clusterer to be used *)
		ipSample	:	ITcUnknown;	(* Container holding a single input sample (ContainerType_Vector_REAL or ContainerType_Vector_LREAL) *)
	END_VAR
	VAR_IN_OUT
		nCluster	:	DINT;	(* Returns the ID of the cluster the sample has been assigned to *)
	END_VAR
	VAR_INPUT
		hrPrev	:	HRESULT;	(* HRESULT indicating the result of previous operations (If SUCCEEDED(hrPrev) equals false, no operation is executed.) *)
	END_VAR

END_FUNCTION

// Functions/Machine Learning/F_VN_GetSampleClusterExp

	{attribute 'TcIecLibraryType'}
	{attribute 'external_name' := 'F_VN_GetSampleClusterExp_GUID_5CE423E8_8BEB_28FB_568B_238558B05B96'}
	(* Get the ID of the best-matching cluster of a single sample. (expert function) *)
	FUNCTION F_VN_GetSampleClusterExp : HRESULT
	VAR_INPUT
		ipClusterer	:	ITcVnMlModel;	(* Clusterer to be used *)
		ipSample	:	ITcUnknown;	(* Container holding a single input sample (ContainerType_Vector_REAL or ContainerType_Vector_LREAL) *)
	END_VAR
	VAR_IN_OUT
		nCluster	:	DINT;	(* Returns the ID of the cluster the sample has been assigned to *)
	END_VAR
	VAR_INPUT
		fNovelty	:	REFERENCE TO REAL;	(* Returns the degree of novelty (0.0 if a sample is completely known; > 0.0 otherwise) of the presented sample (optional, set to 0 if not required) *)
		hrPrev	:	HRESULT;	(* HRESULT indicating the result of previous operations (If SUCCEEDED(hrPrev) equals false, no operation is executed.) *)
	END_VAR

END_FUNCTION

// Functions/Machine Learning/F_VN_GetSampleNovelty

	{attribute 'TcIecLibraryType'}
	{attribute 'external_name' := 'F_VN_GetSampleNovelty_GUID_BA248B66_16F2_208F_541A_BF39E86E39B4'}
	(* Get the degree of novelty of a single sample. *)
	FUNCTION F_VN_GetSampleNovelty : HRESULT
	VAR_INPUT
		ipNoveltyDetector	:	ITcVnMlModel;	(* Novelty detector to be used *)
		ipSample	:	ITcUnknown;	(* Container holding a single input sample (ContainerType_Vector_REAL or ContainerType_Vector_LREAL) *)
	END_VAR
	VAR_IN_OUT
		fNovelty	:	REAL;	(* Returns the degree of novelty (0.0 if a sample is completely known; > 0.0 otherwise) of the presented sample *)
	END_VAR
	VAR_INPUT
		hrPrev	:	HRESULT;	(* HRESULT indicating the result of previous operations (If SUCCEEDED(hrPrev) equals false, no operation is executed.) *)
	END_VAR

END_FUNCTION

// Functions/Machine Learning/F_VN_InverseFeatureScaling

	{attribute 'TcIecLibraryType'}
	{attribute 'external_name' := 'F_VN_InverseFeatureScaling_GUID_7D032692_AB57_24B7_5047_A1FA9877D93F'}
	(* Apply the inverse of feature scaling to one or more sample(s). *)
	FUNCTION F_VN_InverseFeatureScaling : HRESULT
	VAR_INPUT
		ipSamples	:	ITcVnContainer;	(* Container holding one or more input sample(s) (ContainerType_Vector_REAL, ContainerType_Vector_LREAL, ContainerType_Vector_Vector_REAL, or ContainerType_Vector_Vector_LREAL) *)
		ipScales	:	ITcVnContainer;	(* Container with the scaling parameters of each feature (type ContainerType_Vector_REAL or ContainerType_Vector_LREAL). *)
		ipInverseSamples	:	REFERENCE TO ITcVnContainer;	(* Returns the inversed sample(s) using the scaling type and parameters of ipScales. It has the same type of ipSamples. If the same container ipSamples is used, the source data will be replaced. *)
		hrPrev	:	HRESULT;	(* HRESULT indicating the result of previous operations (If SUCCEEDED(hrPrev) equals false, no operation is executed.) *)
	END_VAR

END_FUNCTION

// Functions/Machine Learning/F_VN_InverseFeatureScaling_REAL

	{attribute 'TcIecLibraryType'}
	{attribute 'external_name' := 'F_VN_InverseFeatureScaling_REAL_GUID_918D3948_B2D4_2ABC_48EB_A69EA11F6C28'}
	(* Apply the inverse of feature scaling to a single value. *)
	FUNCTION F_VN_InverseFeatureScaling_REAL : HRESULT
	VAR_INPUT
		fSample	:	REAL;	(* Sample value *)
		ipScales	:	ITcVnContainer;	(* Container with the scaling parameters of each feature (type ContainerType_Vector_REAL or ContainerType_Vector_LREAL). *)
	END_VAR
	VAR_IN_OUT
		fInverseSample	:	REAL;	(* Returns the inversed sample. *)
	END_VAR
	VAR_INPUT
		hrPrev	:	HRESULT;	(* HRESULT indicating the result of previous operations (If SUCCEEDED(hrPrev) equals false, no operation is executed.) *)
	END_VAR

END_FUNCTION

// Functions/Machine Learning/F_VN_InverseFeatureScalingExp

	{attribute 'TcIecLibraryType'}
	{attribute 'external_name' := 'F_VN_InverseFeatureScalingExp_GUID_E39D5E2B_73CD_2834_62B7_A7FA89796173'}
	(* Apply the inverse of feature scaling to one or more sample(s). [fA, fB] should be used if the scaling has been performed using TCVN_FST1_MINMAX with a predetermined output range.. (expert function) *)
	FUNCTION F_VN_InverseFeatureScalingExp : HRESULT
	VAR_INPUT
		ipSamples	:	ITcVnContainer;	(* Container holding one or more input sample(s) (ContainerType_Vector_REAL, ContainerType_Vector_LREAL, ContainerType_Vector_Vector_REAL, or ContainerType_Vector_Vector_LREAL) *)
		ipScales	:	ITcVnContainer;	(* Container with the scaling parameters of each feature (type ContainerType_Vector_REAL or ContainerType_Vector_LREAL). *)
		ipInverseSamples	:	REFERENCE TO ITcVnContainer;	(* Returns the inversed sample(s) using the scaling type and parameters of ipScales. It has the same type of ipSamples. If the same container ipSamples is used, the source data will be replaced. *)
		fA	:	LREAL;	(* represents the lower bound of the range for TCVN_FST1_MINMAX *)
		fB	:	LREAL;	(* represents the upper bound of the range for TCVN_FST1_MINMAX *)
		hrPrev	:	HRESULT;	(* HRESULT indicating the result of previous operations (If SUCCEEDED(hrPrev) equals false, no operation is executed.) *)
	END_VAR

END_FUNCTION

// Functions/Machine Learning/F_VN_InverseFeatureScalingExp_REAL

	{attribute 'TcIecLibraryType'}
	{attribute 'external_name' := 'F_VN_InverseFeatureScalingExp_REAL_GUID_4A3BC586_8A95_2A69_6CA1_8F0151223FC8'}
	(* Apply the inverse of feature scaling to a single value. [fA, fB] should be used if the scaling has been performed using TCVN_FST1_MINMAX with a predetermined output range. *)
	FUNCTION F_VN_InverseFeatureScalingExp_REAL : HRESULT
	VAR_INPUT
		fSample	:	REAL;	(* Sample value *)
		ipScales	:	ITcVnContainer;	(* Container with the scaling parameters of each feature (type ContainerType_Vector_REAL or ContainerType_Vector_LREAL). *)
	END_VAR
	VAR_IN_OUT
		fInverseSample	:	REAL;	(* Returns the inversed sample. *)
	END_VAR
	VAR_INPUT
		fA	:	LREAL;	(* represents the lower bound of the range for TCVN_FST1_MINMAX *)
		fB	:	LREAL;	(* represents the upper bound of the range for TCVN_FST1_MINMAX *)
		hrPrev	:	HRESULT;	(* HRESULT indicating the result of previous operations (If SUCCEEDED(hrPrev) equals false, no operation is executed.) *)
	END_VAR

END_FUNCTION

// Functions/Machine Learning/F_VN_InverseFeatureTransform

	{attribute 'TcIecLibraryType'}
	{attribute 'external_name' := 'F_VN_InverseFeatureTransform_GUID_B576960F_E1D1_2CCE_455A_B74D2EEE326C'}
	(* Apply an inverse feature transform to one or more sample(s). *)
	FUNCTION F_VN_InverseFeatureTransform : HRESULT
	VAR_INPUT
		ipFeatureTransform	:	ITcVnMlModel;	(* Feature transform instance to be used *)
		ipSamples	:	ITcUnknown;	(* Container holding one or more of input sample(s) (ContainerType_Vector_REAL, ContainerType_Vector_LREAL, ContainerType_Vector_Vector_REAL, or ContainerType_Vector_Vector_LREAL) *)
		pipTransformed	:	POINTER TO ITcUnknown;	(* Returns the transformed sample(s) using the same type like ipSamples *)
		hrPrev	:	HRESULT;	(* HRESULT indicating the result of previous operations (If SUCCEEDED(hrPrev) equals false, no operation is executed.) *)
	END_VAR

END_FUNCTION

// Functions/Machine Learning/F_VN_PredictBatch

	{attribute 'TcIecLibraryType'}
	{attribute 'external_name' := 'F_VN_PredictBatch_GUID_FEE60D63_3AB4_2618_6E85_73F6D264EF94'}
	(* Compute predictions for a batch of samples. *)
	FUNCTION F_VN_PredictBatch : HRESULT
	VAR_INPUT
		ipMlModel	:	ITcVnMlModel;	(* Classifier or regressor to be used *)
		ipSamples	:	ITcUnknown;	(* Container holding a batch of input samples (ContainerType_Vector_Vector_REAL or ContainerType_Vector_Vector_LREAL) *)
		ipPredictions	:	REFERENCE TO ITcVnContainer;	(* Returns the predicted outputs (depending on ipSamples; class labels (for classification, ContainerType_Vector_DINT) or real-valued predictions (for regression with scalar output, ContainerType_Vector_REAL or ContainerType_Vector_LREAL; for regression with vectorial output, ContainerType_Vector_Vector_REAL or ContainerType_Vector_Vector_LREAL)) *)
		hrPrev	:	HRESULT;	(* HRESULT indicating the result of previous operations (If SUCCEEDED(hrPrev) equals false, no operation is executed.) *)
	END_VAR

END_FUNCTION

// Functions/Machine Learning/F_VN_PredictBatchExp

	{attribute 'TcIecLibraryType'}
	{attribute 'external_name' := 'F_VN_PredictBatchExp_GUID_400316A8_C606_2201_5BC9_AE0D331EFA15'}
	(* Compute predictions for a batch of samples. (expert function) *)
	FUNCTION F_VN_PredictBatchExp : HRESULT
	VAR_INPUT
		ipMlModel	:	ITcVnMlModel;	(* Classifier or regressor to be used *)
		ipSamples	:	ITcUnknown;	(* Container holding a batch of input samples (ContainerType_Vector_Vector_REAL or ContainerType_Vector_Vector_LREAL) *)
		ipPredictions	:	REFERENCE TO ITcVnContainer;	(* Returns the predicted outputs (depending on ipSamples; class labels (for classification, ContainerType_Vector_DINT) or real-valued predictions (for regression with scalar output, ContainerType_Vector_REAL or ContainerType_Vector_LREAL; for regression with vectorial output, ContainerType_Vector_Vector_REAL or ContainerType_Vector_Vector_LREAL)) *)
		ipNovelties	:	REFERENCE TO ITcVnContainer;	(* Returns the degree of novelty (0.0 if a sample is completely known; > 0.0 otherwise) of each sample (ContainerType_Vector_REAL; optional, set to 0 if not required) *)
		hrPrev	:	HRESULT;	(* HRESULT indicating the result of previous operations (If SUCCEEDED(hrPrev) equals false, no operation is executed.) *)
	END_VAR

END_FUNCTION

// Functions/Machine Learning/F_VN_PredictSampleClass

	{attribute 'TcIecLibraryType'}
	{attribute 'external_name' := 'F_VN_PredictSampleClass_GUID_CD918E25_62A2_25C7_71BA_B6EA99C742D8'}
	(* Classify a single sample. *)
	FUNCTION F_VN_PredictSampleClass : HRESULT
	VAR_INPUT
		ipClassifier	:	ITcVnMlModel;	(* Classifier to be used *)
		ipSample	:	ITcUnknown;	(* Container holding a single input sample (ContainerType_Vector_REAL or ContainerType_Vector_LREAL) *)
	END_VAR
	VAR_IN_OUT
		nClass	:	DINT;	(* Returns the classification result *)
	END_VAR
	VAR_INPUT
		hrPrev	:	HRESULT;	(* HRESULT indicating the result of previous operations (If SUCCEEDED(hrPrev) equals false, no operation is executed.) *)
	END_VAR

END_FUNCTION

// Functions/Machine Learning/F_VN_PredictSampleClassExp

	{attribute 'TcIecLibraryType'}
	{attribute 'external_name' := 'F_VN_PredictSampleClassExp_GUID_F97436F7_E2FC_2E37_4D12_FE61115EC6D7'}
	(* Classify a single sample. (expert function) *)
	FUNCTION F_VN_PredictSampleClassExp : HRESULT
	VAR_INPUT
		ipClassifier	:	ITcVnMlModel;	(* Classifier to be used *)
		ipSample	:	ITcUnknown;	(* Container holding a single input sample (ContainerType_Vector_REAL or ContainerType_Vector_LREAL) *)
	END_VAR
	VAR_IN_OUT
		nClass	:	DINT;	(* Returns the classification result *)
	END_VAR
	VAR_INPUT
		fNovelty	:	REFERENCE TO REAL;	(* Returns the degree of novelty (0.0 if a sample is completely known; > 0.0 otherwise) of the presented sample (optional, set to 0 if not required) *)
		hrPrev	:	HRESULT;	(* HRESULT indicating the result of previous operations (If SUCCEEDED(hrPrev) equals false, no operation is executed.) *)
	END_VAR

END_FUNCTION

// Functions/Machine Learning/F_VN_PredictSampleScalar

	{attribute 'TcIecLibraryType'}
	{attribute 'external_name' := 'F_VN_PredictSampleScalar_GUID_23EAF021_F121_21E0_4CD0_1049E13186C0'}
	(* Compute a scalar prediction for a single sample. *)
	FUNCTION F_VN_PredictSampleScalar : HRESULT
	VAR_INPUT
		ipRegressor	:	ITcVnMlModel;	(* Regressor to be used *)
		ipSample	:	ITcUnknown;	(* Container holding a single input sample (ContainerType_Vector_REAL or ContainerType_Vector_LREAL) *)
	END_VAR
	VAR_IN_OUT
		fPrediction	:	REAL;	(* Returns the predicted output *)
	END_VAR
	VAR_INPUT
		hrPrev	:	HRESULT;	(* HRESULT indicating the result of previous operations (If SUCCEEDED(hrPrev) equals false, no operation is executed.) *)
	END_VAR

END_FUNCTION

// Functions/Machine Learning/F_VN_PredictSampleScalarExp

	{attribute 'TcIecLibraryType'}
	{attribute 'external_name' := 'F_VN_PredictSampleScalarExp_GUID_B19E9B36_E1DC_28A9_6FD1_10AA4147457F'}
	(* Compute a scalar prediction for a single sample. (expert function) *)
	FUNCTION F_VN_PredictSampleScalarExp : HRESULT
	VAR_INPUT
		ipRegressor	:	ITcVnMlModel;	(* Regressor to be used *)
		ipSample	:	ITcUnknown;	(* Container holding a single input sample (ContainerType_Vector_REAL or ContainerType_Vector_LREAL) *)
	END_VAR
	VAR_IN_OUT
		fPrediction	:	REAL;	(* Returns the predicted output *)
	END_VAR
	VAR_INPUT
		fNovelty	:	REFERENCE TO REAL;	(* Returns the degree of novelty (0.0 if a sample is completely known; > 0.0 otherwise) of the presented sample (optional, set to 0 if not required) *)
		hrPrev	:	HRESULT;	(* HRESULT indicating the result of previous operations (If SUCCEEDED(hrPrev) equals false, no operation is executed.) *)
	END_VAR

END_FUNCTION

// Functions/Machine Learning/F_VN_PredictSampleVector

	{attribute 'TcIecLibraryType'}
	{attribute 'external_name' := 'F_VN_PredictSampleVector_GUID_90CD0B30_5A87_25F1_518A_FCE7FFF244B5'}
	(* Compute a vectorial prediction for a single sample. *)
	FUNCTION F_VN_PredictSampleVector : HRESULT
	VAR_INPUT
		ipRegressor	:	ITcVnMlModel;	(* Regressor to be used *)
		ipSample	:	ITcUnknown;	(* Container holding a single input sample (ContainerType_Vector_REAL or ContainerType_Vector_LREAL) *)
		ipPrediction	:	REFERENCE TO ITcVnContainer;	(* Returns the predicted output (ContainerType_Vector_REAL or ContainerType_Vector_LREAL, depending on ipSample) *)
		hrPrev	:	HRESULT;	(* HRESULT indicating the result of previous operations (If SUCCEEDED(hrPrev) equals false, no operation is executed.) *)
	END_VAR

END_FUNCTION

// Functions/Machine Learning/F_VN_PredictSampleVectorExp

	{attribute 'TcIecLibraryType'}
	{attribute 'external_name' := 'F_VN_PredictSampleVectorExp_GUID_8093FEC5_EC0C_2E0A_6D18_81697A93FA5F'}
	(* Compute a vectorial prediction for a single sample. (expert function) *)
	FUNCTION F_VN_PredictSampleVectorExp : HRESULT
	VAR_INPUT
		ipRegressor	:	ITcVnMlModel;	(* Regressor to be used *)
		ipSample	:	ITcUnknown;	(* Container holding a single input sample (ContainerType_Vector_REAL or ContainerType_Vector_LREAL) *)
		ipPrediction	:	REFERENCE TO ITcVnContainer;	(* Returns the predicted output (ContainerType_Vector_REAL or ContainerType_Vector_LREAL, depending on ipSample) *)
		fNovelty	:	REFERENCE TO REAL;	(* Returns the degree of novelty (0.0 if a sample is completely known; > 0.0 otherwise) of the presented sample (optional, set to 0 if not required) *)
		hrPrev	:	HRESULT;	(* HRESULT indicating the result of previous operations (If SUCCEEDED(hrPrev) equals false, no operation is executed.) *)
	END_VAR

END_FUNCTION

// Functions/Machine Learning/F_VN_FeatureScaling

	{attribute 'TcIecLibraryType'}
	{attribute 'external_name' := 'F_VN_FeatureScaling_GUID_18557A89_8D86_2370_761F_86155DCEEB41'}
	(* Apply a feature scaling to one or more sample(s). *)
	FUNCTION F_VN_FeatureScaling : HRESULT
	VAR_INPUT
		ipSamples	:	ITcVnContainer;	(* Container holding one or more input sample(s) (ContainerType_Vector_REAL, ContainerType_Vector_LREAL, ContainerType_Vector_Vector_REAL, or ContainerType_Vector_Vector_LREAL) *)
		ipScales	:	ITcVnContainer;	(* Container with the scaling parameters of each feature (type ContainerType_Vector_REAL or ContainerType_Vector_LREAL). *)
		ipScaledSamples	:	REFERENCE TO ITcVnContainer;	(* Returns the scaled sample(s) using the same type like ipSamples. If the same container ipSamples is uesd, the source data will be replaced. *)
		hrPrev	:	HRESULT;	(* HRESULT indicating the result of previous operations (If SUCCEEDED(hrPrev) equals false, no operation is executed.) *)
	END_VAR

END_FUNCTION

// Functions/Machine Learning/F_VN_FeatureScalingExp

	{attribute 'TcIecLibraryType'}
	{attribute 'external_name' := 'F_VN_FeatureScalingExp_GUID_E152E439_369F_2DFF_5BDE_CA3EA6C1915D'}
	(* Apply a feature scaling to one or more sample(s) and get output range between [fA, fB] in the case of TCVN_FST1_MINMAX.  (expert function) *)
	FUNCTION F_VN_FeatureScalingExp : HRESULT
	VAR_INPUT
		ipSamples	:	ITcVnContainer;	(* Container holding one or more input sample(s) (ContainerType_Vector_REAL, ContainerType_Vector_LREAL, ContainerType_Vector_Vector_REAL, or ContainerType_Vector_Vector_LREAL) *)
		ipScales	:	ITcVnContainer;	(* Container with the scaling parameters of each feature (type ContainerType_Vector_REAL or ContainerType_Vector_LREAL). *)
		ipScaledSamples	:	REFERENCE TO ITcVnContainer;	(* Returns the scaled sample(s) using the same type like ipSamples. If the same container ipSamples is uesd, the source data will be replaced. *)
		fA	:	LREAL;	(* represents the lower bound of the range for TCVN_FST1_MINMAX *)
		fB	:	LREAL;	(* represents the upper bound of the range for TCVN_FST1_MINMAX *)
		hrPrev	:	HRESULT;	(* HRESULT indicating the result of previous operations (If SUCCEEDED(hrPrev) equals false, no operation is executed.) *)
	END_VAR

END_FUNCTION

// Functions/Machine Learning/F_VN_TrainBatch

	{attribute 'TcIecLibraryType'}
	{attribute 'external_name' := 'F_VN_TrainBatch_GUID_F41885E6_DF63_2CD8_63C1_ED4B9835C0A5'}
	(* Train a classifier, a clusterer, a novelty detector, or a regressor with a batch of samples. On-line trainable models are trained once with each sample. Depending on the application and the number of available training samples, repeated training of such models with the same data may improve the results. *)
	FUNCTION F_VN_TrainBatch : HRESULT
	VAR_INPUT
		ipMlModel	:	ITcVnMlModel;	(* Classifier, clusterer, novelty detector, or regressor to be used *)
		ipSamples	:	ITcUnknown;	(* Container holding a batch of input samples (ContainerType_Vector_Vector_REAL or ContainerType_Vector_Vector_LREAL) *)
		ipOutputs	:	ITcVnContainer;	(* Class labels (for classification, ContainerType_Vector_DINT) or target outputs (for regression with scalar output, ContainerType_Vector_REAL or ContainerType_Vector_LREAL; for regression with vectorial output, ContainerType_Vector_Vector_REAL or ContainerType_Vector_Vector_LREAL) to be learnt (must be 0 for clusterers and for novelty detectors) *)
		hrPrev	:	HRESULT;	(* HRESULT indicating the result of previous operations (If SUCCEEDED(hrPrev) equals false, no operation is executed.) *)
	END_VAR

END_FUNCTION

// Functions/Machine Learning/F_VN_TrainBatchClusters

	{attribute 'TcIecLibraryType'}
	{attribute 'external_name' := 'F_VN_TrainBatchClusters_GUID_A0CA738D_F363_2818_50A9_558458A7B718'}
	(* Train a clusterer with a batch of samples and return the IDs of the clusters the samples have been assigned to, if requested. On-line trainable clusterers are trained once with each sample. Depending on the application and the number of available training samples, repeated training of such models with the same data may improve the results. *)
	FUNCTION F_VN_TrainBatchClusters : HRESULT
	VAR_INPUT
		ipClusterer	:	ITcVnMlModel;	(* Clusterer to be used *)
		ipSamples	:	ITcUnknown;	(* Container holding a batch of input samples (ContainerType_Vector_Vector_REAL or ContainerType_Vector_Vector_LREAL) *)
		ipClusters	:	REFERENCE TO ITcVnContainer;	(* Returns the IDs of the clusters the samples have been assigned to (ContainerType_Vector_DINT; optional, set to 0 if not required) *)
		hrPrev	:	HRESULT;	(* HRESULT indicating the result of previous operations (If SUCCEEDED(hrPrev) equals false, no operation is executed.) *)
	END_VAR

END_FUNCTION

// Functions/Machine Learning/F_VN_TrainSample

	{attribute 'TcIecLibraryType'}
	{attribute 'external_name' := 'F_VN_TrainSample_GUID_E886DF26_903C_2C12_52C7_577977C55CAE'}
	(* Train a clusterer or a novelty detector with a single sample. *)
	FUNCTION F_VN_TrainSample : HRESULT
	VAR_INPUT
		ipMlModel	:	ITcVnMlModel;	(* Clusterer or novelty detector to be used *)
		ipSample	:	ITcUnknown;	(* Container holding a single input sample (ContainerType_Vector_REAL or ContainerType_Vector_LREAL) *)
		hrPrev	:	HRESULT;	(* HRESULT indicating the result of previous operations (If SUCCEEDED(hrPrev) equals false, no operation is executed.) *)
	END_VAR

END_FUNCTION

// Functions/Machine Learning/F_VN_TrainSampleClass

	{attribute 'TcIecLibraryType'}
	{attribute 'external_name' := 'F_VN_TrainSampleClass_GUID_8246E157_F354_2D63_5479_1130EEB0E23C'}
	(* Train a classifier with a single sample. *)
	FUNCTION F_VN_TrainSampleClass : HRESULT
	VAR_INPUT
		ipClassifier	:	ITcVnMlModel;	(* Classifier to be used *)
		ipSample	:	ITcUnknown;	(* Container holding a single input sample (ContainerType_Vector_REAL or ContainerType_Vector_LREAL) *)
		nClass	:	DINT;	(* Class label to be learnt *)
		hrPrev	:	HRESULT;	(* HRESULT indicating the result of previous operations (If SUCCEEDED(hrPrev) equals false, no operation is executed.) *)
	END_VAR

END_FUNCTION

// Functions/Machine Learning/F_VN_TrainSampleCluster

	{attribute 'TcIecLibraryType'}
	{attribute 'external_name' := 'F_VN_TrainSampleCluster_GUID_B3DECB05_78F8_29E9_5CC3_C3675043D266'}
	(* Train a clusterer with a single sample and return the ID of the cluster the sample has been assigned to, if requested. The clusterer must be online trainable. *)
	FUNCTION F_VN_TrainSampleCluster : HRESULT
	VAR_INPUT
		ipClusterer	:	ITcVnMlModel;	(* Clusterer to be used *)
		ipSample	:	ITcUnknown;	(* Container holding a single input sample (ContainerType_Vector_REAL or ContainerType_Vector_LREAL) *)
		nCluster	:	REFERENCE TO DINT;	(* Returns the ID of the cluster the sample has been assigned to (If the pointer is 0, no cluster ID is requested.) *)
		hrPrev	:	HRESULT;	(* HRESULT indicating the result of previous operations (If SUCCEEDED(hrPrev) equals false, no operation is executed.) *)
	END_VAR

END_FUNCTION

// Functions/Machine Learning/F_VN_TrainSampleScalar

	{attribute 'TcIecLibraryType'}
	{attribute 'external_name' := 'F_VN_TrainSampleScalar_GUID_DB5DAD42_261E_223A_5EE1_261928227C1E'}
	(* Train a regressor with a single sample and scalar output. *)
	FUNCTION F_VN_TrainSampleScalar : HRESULT
	VAR_INPUT
		ipRegressor	:	ITcVnMlModel;	(* Regressor to be used *)
		ipSample	:	ITcUnknown;	(* Container holding a single input sample (ContainerType_Vector_REAL or ContainerType_Vector_LREAL) *)
		fOutput	:	REAL;	(* Scalar output to be learnt *)
		hrPrev	:	HRESULT;	(* HRESULT indicating the result of previous operations (If SUCCEEDED(hrPrev) equals false, no operation is executed.) *)
	END_VAR

END_FUNCTION

// Functions/Machine Learning/F_VN_TrainSampleVector

	{attribute 'TcIecLibraryType'}
	{attribute 'external_name' := 'F_VN_TrainSampleVector_GUID_2206E11B_0B9A_2903_5377_29F300E94755'}
	(* Train a regressor with a single sample and vectorial output. *)
	FUNCTION F_VN_TrainSampleVector : HRESULT
	VAR_INPUT
		ipRegressor	:	ITcVnMlModel;	(* Regressor to be used *)
		ipSample	:	ITcUnknown;	(* Container holding a single input sample (ContainerType_Vector_REAL or ContainerType_Vector_LREAL) *)
		ipOutput	:	ITcVnContainer;	(* Vectorial output to be learnt (ContainerType_Vector_REAL or ContainerType_Vector_LREAL) *)
		hrPrev	:	HRESULT;	(* HRESULT indicating the result of previous operations (If SUCCEEDED(hrPrev) equals false, no operation is executed.) *)
	END_VAR

END_FUNCTION

// Functions/Drawing/F_VN_DrawArrow

